REGION Network 5: Call production data cycle timer
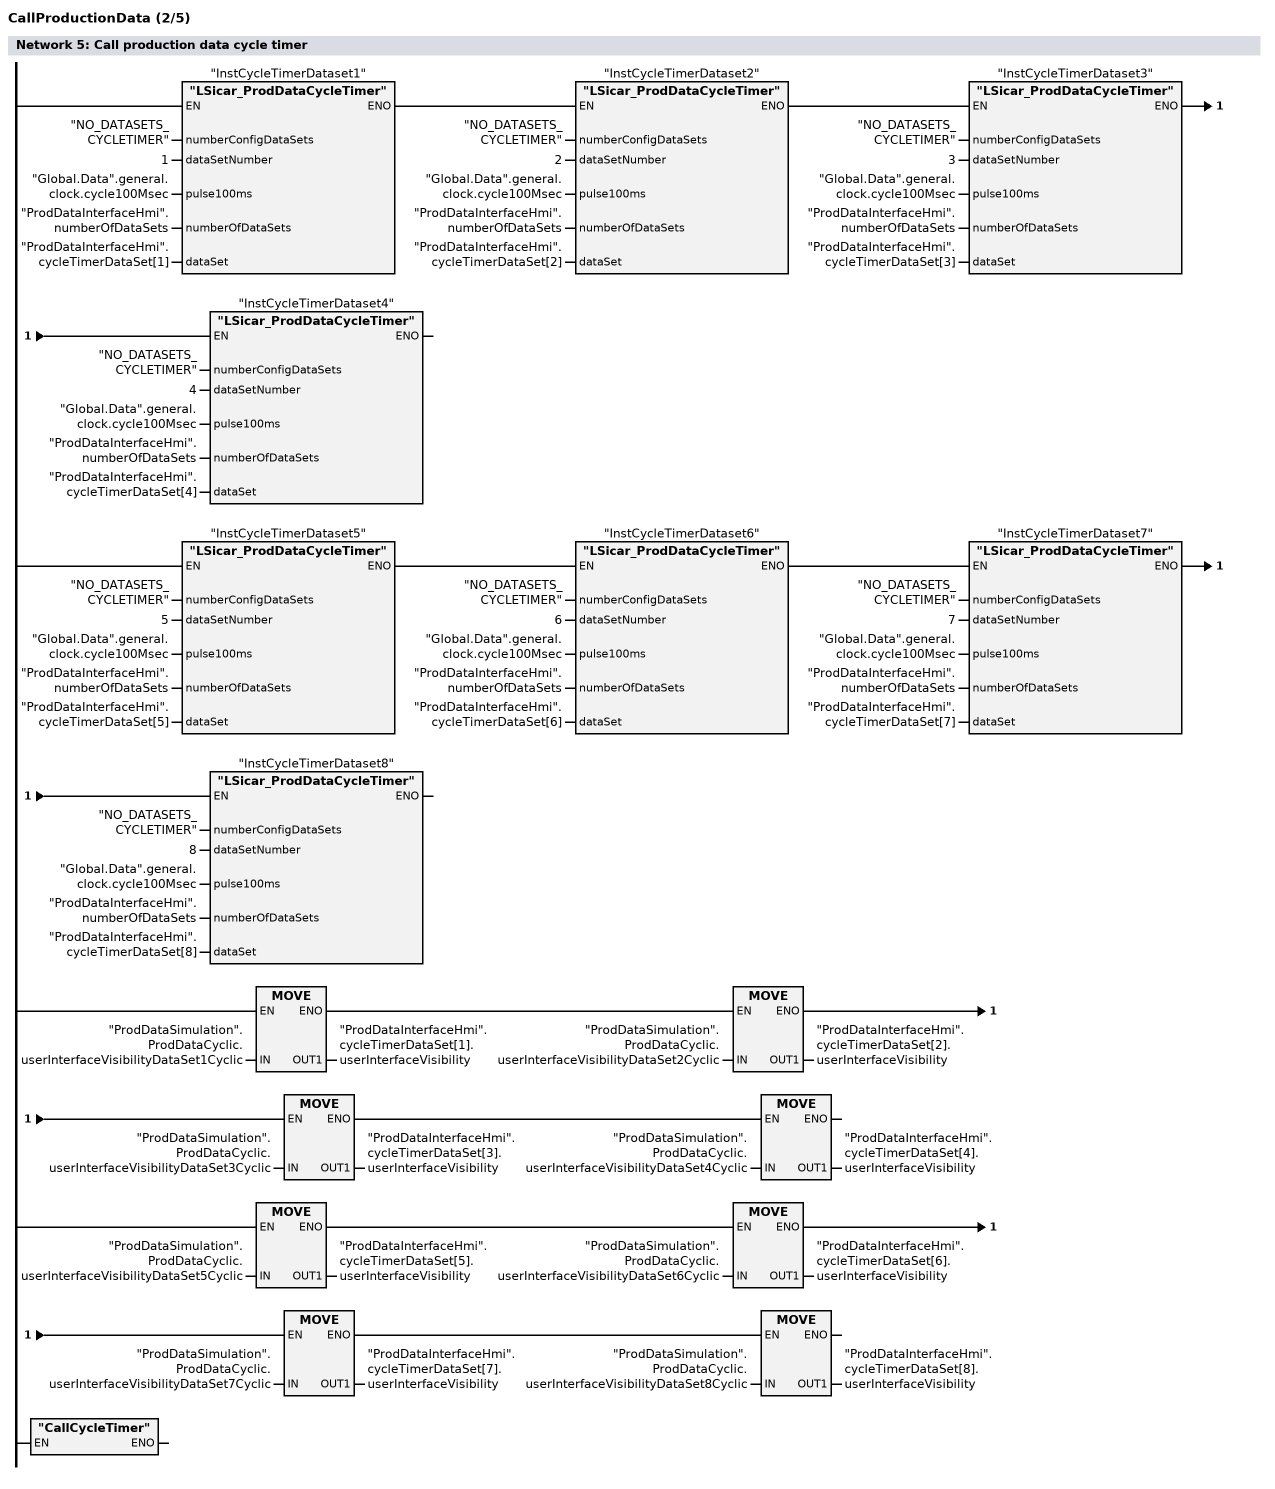
   RUNG wire#powerrail
      "InstCycleTimerDataset1"(numberConfigDataSets := "NO_DATASETS_CYCLETIMER", dataSetNumber := 1, pulse100ms := "Global.Data".general.clock.cycle100Msec, numberOfDataSets := "ProdDataInterfaceHmi".numberOfDataSets, dataSet := "ProdDataInterfaceHmi".cycleTimerDataSet[1])
      "InstCycleTimerDataset2"(numberConfigDataSets := "NO_DATASETS_CYCLETIMER", dataSetNumber := 2, pulse100ms := "Global.Data".general.clock.cycle100Msec, numberOfDataSets := "ProdDataInterfaceHmi".numberOfDataSets, dataSet := "ProdDataInterfaceHmi".cycleTimerDataSet[2])
      "InstCycleTimerDataset3"(numberConfigDataSets := "NO_DATASETS_CYCLETIMER", dataSetNumber := 3, pulse100ms := "Global.Data".general.clock.cycle100Msec, numberOfDataSets := "ProdDataInterfaceHmi".numberOfDataSets, dataSet := "ProdDataInterfaceHmi".cycleTimerDataSet[3])
      "InstCycleTimerDataset4"(numberConfigDataSets := "NO_DATASETS_CYCLETIMER", dataSetNumber := 4, pulse100ms := "Global.Data".general.clock.cycle100Msec, numberOfDataSets := "ProdDataInterfaceHmi".numberOfDataSets, dataSet := "ProdDataInterfaceHmi".cycleTimerDataSet[4])
   END_RUNG
   RUNG wire#powerrail
      "InstCycleTimerDataset5"(numberConfigDataSets := "NO_DATASETS_CYCLETIMER", dataSetNumber := 5, pulse100ms := "Global.Data".general.clock.cycle100Msec, numberOfDataSets := "ProdDataInterfaceHmi".numberOfDataSets, dataSet := "ProdDataInterfaceHmi".cycleTimerDataSet[5])
      "InstCycleTimerDataset6"(numberConfigDataSets := "NO_DATASETS_CYCLETIMER", dataSetNumber := 6, pulse100ms := "Global.Data".general.clock.cycle100Msec, numberOfDataSets := "ProdDataInterfaceHmi".numberOfDataSets, dataSet := "ProdDataInterfaceHmi".cycleTimerDataSet[6])
      "InstCycleTimerDataset7"(numberConfigDataSets := "NO_DATASETS_CYCLETIMER", dataSetNumber := 7, pulse100ms := "Global.Data".general.clock.cycle100Msec, numberOfDataSets := "ProdDataInterfaceHmi".numberOfDataSets, dataSet := "ProdDataInterfaceHmi".cycleTimerDataSet[7])
      "InstCycleTimerDataset8"(numberConfigDataSets := "NO_DATASETS_CYCLETIMER", dataSetNumber := 8, pulse100ms := "Global.Data".general.clock.cycle100Msec, numberOfDataSets := "ProdDataInterfaceHmi".numberOfDataSets, dataSet := "ProdDataInterfaceHmi".cycleTimerDataSet[8])
   END_RUNG
   RUNG wire#powerrail
      Move(in := "ProdDataSimulation".ProdDataCyclic.userInterfaceVisibilityDataSet1Cyclic, out1 => "ProdDataInterfaceHmi".cycleTimerDataSet[1].userInterfaceVisibility)
      Move(in := "ProdDataSimulation".ProdDataCyclic.userInterfaceVisibilityDataSet2Cyclic, out1 => "ProdDataInterfaceHmi".cycleTimerDataSet[2].userInterfaceVisibility)
      Move(in := "ProdDataSimulation".ProdDataCyclic.userInterfaceVisibilityDataSet3Cyclic, out1 => "ProdDataInterfaceHmi".cycleTimerDataSet[3].userInterfaceVisibility)
      Move(in := "ProdDataSimulation".ProdDataCyclic.userInterfaceVisibilityDataSet4Cyclic, out1 => "ProdDataInterfaceHmi".cycleTimerDataSet[4].userInterfaceVisibility)
   END_RUNG
   RUNG wire#powerrail
      Move(in := "ProdDataSimulation".ProdDataCyclic.userInterfaceVisibilityDataSet5Cyclic, out1 => "ProdDataInterfaceHmi".cycleTimerDataSet[5].userInterfaceVisibility)
      Move(in := "ProdDataSimulation".ProdDataCyclic.userInterfaceVisibilityDataSet6Cyclic, out1 => "ProdDataInterfaceHmi".cycleTimerDataSet[6].userInterfaceVisibility)
      Move(in := "ProdDataSimulation".ProdDataCyclic.userInterfaceVisibilityDataSet7Cyclic, out1 => "ProdDataInterfaceHmi".cycleTimerDataSet[7].userInterfaceVisibility)
      Move(in := "ProdDataSimulation".ProdDataCyclic.userInterfaceVisibilityDataSet8Cyclic, out1 => "ProdDataInterfaceHmi".cycleTimerDataSet[8].userInterfaceVisibility)
   END_RUNG
   RUNG wire#powerrail
      "CallCycleTimer"()
   END_RUNG
   // the same network as SCL:
   "InstCycleTimerDataset1"(numberConfigDataSets := "NO_DATASETS_CYCLETIMER",   // "LSicar_ProdDataCycleTimer"
                           dataSetNumber := 1,
                           pulse100ms := "Global.Data".general.clock.cycle100Msec,
                           numberOfDataSets := "ProdDataInterfaceHmi".numberOfDataSets,
                           dataSet := "ProdDataInterfaceHmi".cycleTimerDataSet[1],
                           ENO => #_w1);
   "InstCycleTimerDataset2"(EN := #_w1,   // "LSicar_ProdDataCycleTimer"
                           numberConfigDataSets := "NO_DATASETS_CYCLETIMER",
                           dataSetNumber := 2,
                           pulse100ms := "Global.Data".general.clock.cycle100Msec,
                           numberOfDataSets := "ProdDataInterfaceHmi".numberOfDataSets,
                           dataSet := "ProdDataInterfaceHmi".cycleTimerDataSet[2],
                           ENO => #_w2);
   "InstCycleTimerDataset3"(EN := #_w2,   // "LSicar_ProdDataCycleTimer"
                           numberConfigDataSets := "NO_DATASETS_CYCLETIMER",
                           dataSetNumber := 3,
                           pulse100ms := "Global.Data".general.clock.cycle100Msec,
                           numberOfDataSets := "ProdDataInterfaceHmi".numberOfDataSets,
                           dataSet := "ProdDataInterfaceHmi".cycleTimerDataSet[3],
                           ENO => #_w3);
   IF #_w3 THEN
       "InstCycleTimerDataset4"(numberConfigDataSets := "NO_DATASETS_CYCLETIMER",   // "LSicar_ProdDataCycleTimer"
                               dataSetNumber := 4,
                               pulse100ms := "Global.Data".general.clock.cycle100Msec,
                               numberOfDataSets := "ProdDataInterfaceHmi".numberOfDataSets,
                               dataSet := "ProdDataInterfaceHmi".cycleTimerDataSet[4]);
   END_IF;
   "InstCycleTimerDataset5"(numberConfigDataSets := "NO_DATASETS_CYCLETIMER",   // "LSicar_ProdDataCycleTimer"
                           dataSetNumber := 5,
                           pulse100ms := "Global.Data".general.clock.cycle100Msec,
                           numberOfDataSets := "ProdDataInterfaceHmi".numberOfDataSets,
                           dataSet := "ProdDataInterfaceHmi".cycleTimerDataSet[5],
                           ENO => #_w4);
   "InstCycleTimerDataset6"(EN := #_w4,   // "LSicar_ProdDataCycleTimer"
                           numberConfigDataSets := "NO_DATASETS_CYCLETIMER",
                           dataSetNumber := 6,
                           pulse100ms := "Global.Data".general.clock.cycle100Msec,
                           numberOfDataSets := "ProdDataInterfaceHmi".numberOfDataSets,
                           dataSet := "ProdDataInterfaceHmi".cycleTimerDataSet[6],
                           ENO => #_w5);
   "InstCycleTimerDataset7"(EN := #_w5,   // "LSicar_ProdDataCycleTimer"
                           numberConfigDataSets := "NO_DATASETS_CYCLETIMER",
                           dataSetNumber := 7,
                           pulse100ms := "Global.Data".general.clock.cycle100Msec,
                           numberOfDataSets := "ProdDataInterfaceHmi".numberOfDataSets,
                           dataSet := "ProdDataInterfaceHmi".cycleTimerDataSet[7],
                           ENO => #_w6);
   IF #_w6 THEN
       "InstCycleTimerDataset8"(numberConfigDataSets := "NO_DATASETS_CYCLETIMER",   // "LSicar_ProdDataCycleTimer"
                               dataSetNumber := 8,
                               pulse100ms := "Global.Data".general.clock.cycle100Msec,
                               numberOfDataSets := "ProdDataInterfaceHmi".numberOfDataSets,
                               dataSet := "ProdDataInterfaceHmi".cycleTimerDataSet[8]);
   END_IF;
   "ProdDataInterfaceHmi".cycleTimerDataSet[1].userInterfaceVisibility := "ProdDataSimulation".ProdDataCyclic.userInterfaceVisibilityDataSet1Cyclic;
   "ProdDataInterfaceHmi".cycleTimerDataSet[2].userInterfaceVisibility := "ProdDataSimulation".ProdDataCyclic.userInterfaceVisibilityDataSet2Cyclic;
   "ProdDataInterfaceHmi".cycleTimerDataSet[3].userInterfaceVisibility := "ProdDataSimulation".ProdDataCyclic.userInterfaceVisibilityDataSet3Cyclic;
   "ProdDataInterfaceHmi".cycleTimerDataSet[4].userInterfaceVisibility := "ProdDataSimulation".ProdDataCyclic.userInterfaceVisibilityDataSet4Cyclic;
   "ProdDataInterfaceHmi".cycleTimerDataSet[5].userInterfaceVisibility := "ProdDataSimulation".ProdDataCyclic.userInterfaceVisibilityDataSet5Cyclic;
   "ProdDataInterfaceHmi".cycleTimerDataSet[6].userInterfaceVisibility := "ProdDataSimulation".ProdDataCyclic.userInterfaceVisibilityDataSet6Cyclic;
   "ProdDataInterfaceHmi".cycleTimerDataSet[7].userInterfaceVisibility := "ProdDataSimulation".ProdDataCyclic.userInterfaceVisibilityDataSet7Cyclic;
   "ProdDataInterfaceHmi".cycleTimerDataSet[8].userInterfaceVisibility := "ProdDataSimulation".ProdDataCyclic.userInterfaceVisibilityDataSet8Cyclic;
   "CallCycleTimer"();
END_REGION

REGION Network 6: Beispiel: Limit Value 1..2 / Call production data limit values
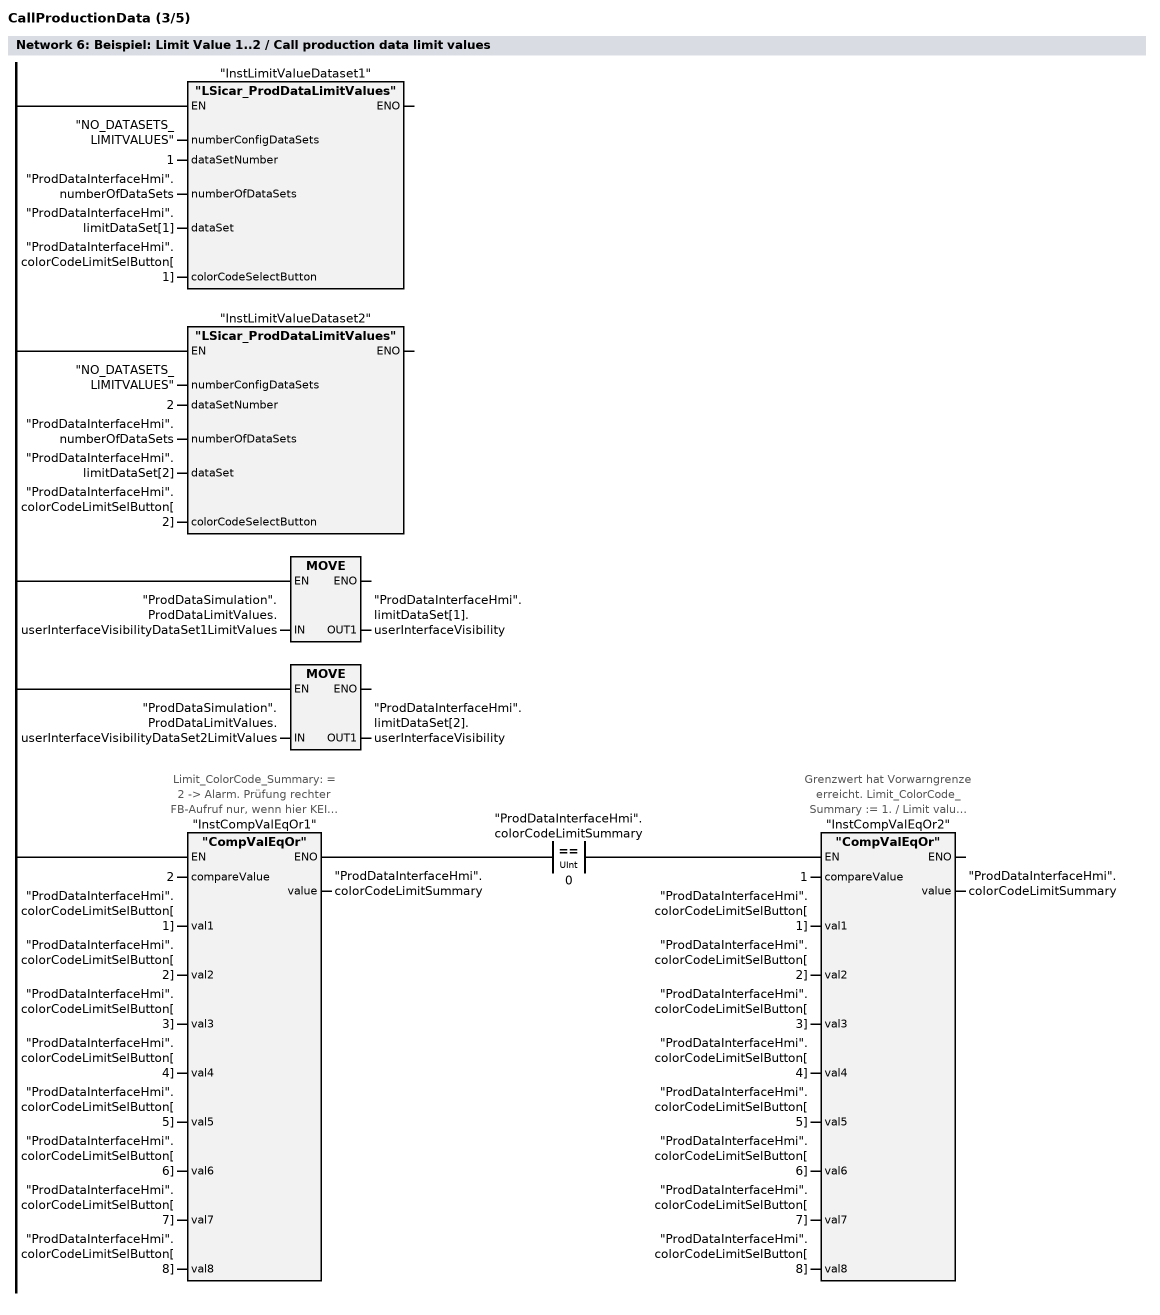
   RUNG wire#powerrail
      "InstLimitValueDataset1"(numberConfigDataSets := "NO_DATASETS_LIMITVALUES", dataSetNumber := 1, numberOfDataSets := "ProdDataInterfaceHmi".numberOfDataSets, dataSet := "ProdDataInterfaceHmi".limitDataSet[1], colorCodeSelectButton := "ProdDataInterfaceHmi".colorCodeLimitSelButton[1])
   END_RUNG
   RUNG wire#powerrail
      "InstLimitValueDataset2"(numberConfigDataSets := "NO_DATASETS_LIMITVALUES", dataSetNumber := 2, numberOfDataSets := "ProdDataInterfaceHmi".numberOfDataSets, dataSet := "ProdDataInterfaceHmi".limitDataSet[2], colorCodeSelectButton := "ProdDataInterfaceHmi".colorCodeLimitSelButton[2])
   END_RUNG
   RUNG wire#powerrail
      Move(in := "ProdDataSimulation".ProdDataLimitValues.userInterfaceVisibilityDataSet1LimitValues, out1 => "ProdDataInterfaceHmi".limitDataSet[1].userInterfaceVisibility)
   END_RUNG
   RUNG wire#powerrail
      Move(in := "ProdDataSimulation".ProdDataLimitValues.userInterfaceVisibilityDataSet2LimitValues, out1 => "ProdDataInterfaceHmi".limitDataSet[2].userInterfaceVisibility)
   END_RUNG
   RUNG wire#powerrail
      "InstCompValEqOr1"(compareValue := 2, val1 := "ProdDataInterfaceHmi".colorCodeLimitSelButton[1], val2 := "ProdDataInterfaceHmi".colorCodeLimitSelButton[2], val3 := "ProdDataInterfaceHmi".colorCodeLimitSelButton[3], val4 := "ProdDataInterfaceHmi".colorCodeLimitSelButton[4], val5 := "ProdDataInterfaceHmi".colorCodeLimitSelButton[5], val6 := "ProdDataInterfaceHmi".colorCodeLimitSelButton[6], val7 := "ProdDataInterfaceHmi".colorCodeLimitSelButton[7], val8 := "ProdDataInterfaceHmi".colorCodeLimitSelButton[8], value => "ProdDataInterfaceHmi".colorCodeLimitSummary)   // Limit_ColorCode_Summary: = 2 -> Alarm. Prüfung rechter FB-Aufruf nur, wenn hier KEIN Alarm (VALUE = 0) ansteht; Alarm ist höher prior. / Limit value = 2 -> Alarm. Limit_ColorCode_Summary := 2. Call right block only, if NO alarm (VALUE = 0) is pending here; alarm is higher prior.
      { S7_Templates := "SrcType := UInt" } EQ_Contact(in1 := "ProdDataInterfaceHmi".colorCodeLimitSummary, in2 := 0)
      "InstCompValEqOr2"(compareValue := 1, val1 := "ProdDataInterfaceHmi".colorCodeLimitSelButton[1], val2 := "ProdDataInterfaceHmi".colorCodeLimitSelButton[2], val3 := "ProdDataInterfaceHmi".colorCodeLimitSelButton[3], val4 := "ProdDataInterfaceHmi".colorCodeLimitSelButton[4], val5 := "ProdDataInterfaceHmi".colorCodeLimitSelButton[5], val6 := "ProdDataInterfaceHmi".colorCodeLimitSelButton[6], val7 := "ProdDataInterfaceHmi".colorCodeLimitSelButton[7], val8 := "ProdDataInterfaceHmi".colorCodeLimitSelButton[8], value => "ProdDataInterfaceHmi".colorCodeLimitSummary)   // Grenzwert hat Vorwarngrenze erreicht. Limit_ColorCode_Summary := 1. / Limit value <= Prewarn value. Limit_ColorCode_Summary := 1.
   END_RUNG
   // the same network as SCL:
   "InstLimitValueDataset1"(numberConfigDataSets := "NO_DATASETS_LIMITVALUES",   // "LSicar_ProdDataLimitValues"
                           dataSetNumber := 1,
                           numberOfDataSets := "ProdDataInterfaceHmi".numberOfDataSets,
                           dataSet := "ProdDataInterfaceHmi".limitDataSet[1],
                           colorCodeSelectButton := "ProdDataInterfaceHmi".colorCodeLimitSelButton[1]);
   "InstLimitValueDataset2"(numberConfigDataSets := "NO_DATASETS_LIMITVALUES",   // "LSicar_ProdDataLimitValues"
                           dataSetNumber := 2,
                           numberOfDataSets := "ProdDataInterfaceHmi".numberOfDataSets,
                           dataSet := "ProdDataInterfaceHmi".limitDataSet[2],
                           colorCodeSelectButton := "ProdDataInterfaceHmi".colorCodeLimitSelButton[2]);
   "ProdDataInterfaceHmi".limitDataSet[1].userInterfaceVisibility := "ProdDataSimulation".ProdDataLimitValues.userInterfaceVisibilityDataSet1LimitValues;
   "ProdDataInterfaceHmi".limitDataSet[2].userInterfaceVisibility := "ProdDataSimulation".ProdDataLimitValues.userInterfaceVisibilityDataSet2LimitValues;
   "InstCompValEqOr1"(compareValue := 2,   // "CompValEqOr": Limit_ColorCode_Summary: = 2 -> Alarm. Prüfung rechter FB-Aufruf nur, wenn hier KEIN Alarm (VALUE = 0) ansteht; Alarm ist höher prior. / Limit value = 2 -> Alarm. Limit_ColorCode_Summary := 2. Call right block only, if NO alarm (VALUE = 0) is pending here; alarm is higher prior.
                      val1 := "ProdDataInterfaceHmi".colorCodeLimitSelButton[1],
                      val2 := "ProdDataInterfaceHmi".colorCodeLimitSelButton[2],
                      val3 := "ProdDataInterfaceHmi".colorCodeLimitSelButton[3],
                      val4 := "ProdDataInterfaceHmi".colorCodeLimitSelButton[4],
                      val5 := "ProdDataInterfaceHmi".colorCodeLimitSelButton[5],
                      val6 := "ProdDataInterfaceHmi".colorCodeLimitSelButton[6],
                      val7 := "ProdDataInterfaceHmi".colorCodeLimitSelButton[7],
                      val8 := "ProdDataInterfaceHmi".colorCodeLimitSelButton[8],
                      value => "ProdDataInterfaceHmi".colorCodeLimitSummary,
                      ENO => #_w1);
   IF #_w1 AND ("ProdDataInterfaceHmi".colorCodeLimitSummary = 0) THEN
       "InstCompValEqOr2"(compareValue := 1,   // "CompValEqOr": Grenzwert hat Vorwarngrenze erreicht. Limit_ColorCode_Summary := 1. / Limit value <= Prewarn value. Limit_ColorCode_Summary := 1.
                          val1 := "ProdDataInterfaceHmi".colorCodeLimitSelButton[1],
                          val2 := "ProdDataInterfaceHmi".colorCodeLimitSelButton[2],
                          val3 := "ProdDataInterfaceHmi".colorCodeLimitSelButton[3],
                          val4 := "ProdDataInterfaceHmi".colorCodeLimitSelButton[4],
                          val5 := "ProdDataInterfaceHmi".colorCodeLimitSelButton[5],
                          val6 := "ProdDataInterfaceHmi".colorCodeLimitSelButton[6],
                          val7 := "ProdDataInterfaceHmi".colorCodeLimitSelButton[7],
                          val8 := "ProdDataInterfaceHmi".colorCodeLimitSelButton[8],
                          value => "ProdDataInterfaceHmi".colorCodeLimitSummary);
   END_IF;
END_REGION

REGION Network 7: Beispiel: Shift Counter 1..2 / Call production data shift counter
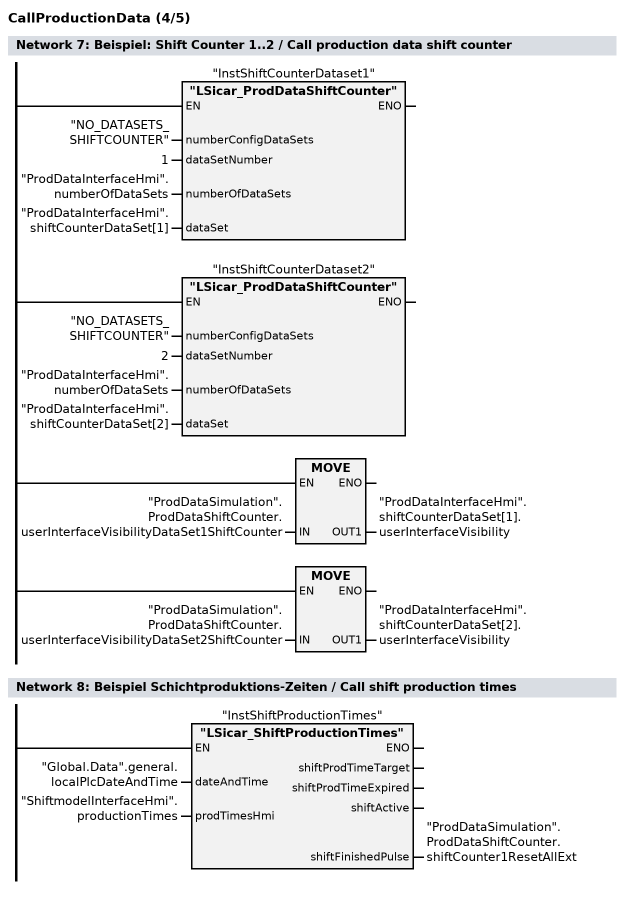
   RUNG wire#powerrail
      "InstShiftCounterDataset1"(numberConfigDataSets := "NO_DATASETS_SHIFTCOUNTER", dataSetNumber := 1, numberOfDataSets := "ProdDataInterfaceHmi".numberOfDataSets, dataSet := "ProdDataInterfaceHmi".shiftCounterDataSet[1])
   END_RUNG
   RUNG wire#powerrail
      "InstShiftCounterDataset2"(numberConfigDataSets := "NO_DATASETS_SHIFTCOUNTER", dataSetNumber := 2, numberOfDataSets := "ProdDataInterfaceHmi".numberOfDataSets, dataSet := "ProdDataInterfaceHmi".shiftCounterDataSet[2])
   END_RUNG
   RUNG wire#powerrail
      Move(in := "ProdDataSimulation".ProdDataShiftCounter.userInterfaceVisibilityDataSet1ShiftCounter, out1 => "ProdDataInterfaceHmi".shiftCounterDataSet[1].userInterfaceVisibility)
   END_RUNG
   RUNG wire#powerrail
      Move(in := "ProdDataSimulation".ProdDataShiftCounter.userInterfaceVisibilityDataSet2ShiftCounter, out1 => "ProdDataInterfaceHmi".shiftCounterDataSet[2].userInterfaceVisibility)
   END_RUNG
   // the same network as SCL:
   "InstShiftCounterDataset1"(numberConfigDataSets := "NO_DATASETS_SHIFTCOUNTER",   // "LSicar_ProdDataShiftCounter"
                           dataSetNumber := 1,
                           numberOfDataSets := "ProdDataInterfaceHmi".numberOfDataSets,
                           dataSet := "ProdDataInterfaceHmi".shiftCounterDataSet[1]);
   "InstShiftCounterDataset2"(numberConfigDataSets := "NO_DATASETS_SHIFTCOUNTER",   // "LSicar_ProdDataShiftCounter"
                           dataSetNumber := 2,
                           numberOfDataSets := "ProdDataInterfaceHmi".numberOfDataSets,
                           dataSet := "ProdDataInterfaceHmi".shiftCounterDataSet[2]);
   "ProdDataInterfaceHmi".shiftCounterDataSet[1].userInterfaceVisibility := "ProdDataSimulation".ProdDataShiftCounter.userInterfaceVisibilityDataSet1ShiftCounter;
   "ProdDataInterfaceHmi".shiftCounterDataSet[2].userInterfaceVisibility := "ProdDataSimulation".ProdDataShiftCounter.userInterfaceVisibilityDataSet2ShiftCounter;
END_REGION

REGION Network 8: Beispiel Schichtproduktions-Zeiten / Call shift production times
   RUNG wire#powerrail
      "InstShiftProductionTimes"(dateAndTime := "Global.Data".general.localPlcDateAndTime, prodTimesHmi := "ShiftmodelInterfaceHmi".productionTimes, shiftProdTimeTarget =>, shiftProdTimeExpired =>, shiftActive =>, shiftFinishedPulse => "ProdDataSimulation".ProdDataShiftCounter.shiftCounter1ResetAllExt)
   END_RUNG
   // the same network as SCL:
   "InstShiftProductionTimes"(dateAndTime := "Global.Data".general.localPlcDateAndTime,   // "LSicar_ShiftProductionTimes"
                           prodTimesHmi := "ShiftmodelInterfaceHmi".productionTimes,
                           shiftFinishedPulse => "ProdDataSimulation".ProdDataShiftCounter.shiftCounter1ResetAllExt);
END_REGION

REGION Network 9: Beispiel: Shift Counter 1..2 + OEE + Trend / Call production data shift counter OEE
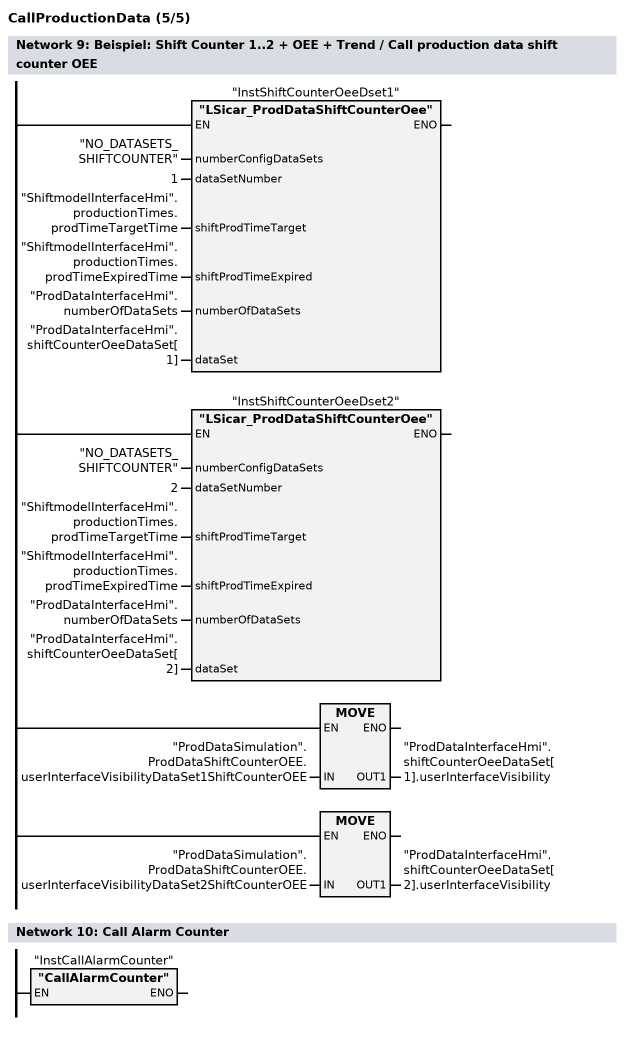
   RUNG wire#powerrail
      "InstShiftCounterOeeDset1"(numberConfigDataSets := "NO_DATASETS_SHIFTCOUNTER", dataSetNumber := 1, shiftProdTimeTarget := "ShiftmodelInterfaceHmi".productionTimes.prodTimeTargetTime, shiftProdTimeExpired := "ShiftmodelInterfaceHmi".productionTimes.prodTimeExpiredTime, numberOfDataSets := "ProdDataInterfaceHmi".numberOfDataSets, dataSet := "ProdDataInterfaceHmi".shiftCounterOeeDataSet[1])
   END_RUNG
   RUNG wire#powerrail
      "InstShiftCounterOeeDset2"(numberConfigDataSets := "NO_DATASETS_SHIFTCOUNTER", dataSetNumber := 2, shiftProdTimeTarget := "ShiftmodelInterfaceHmi".productionTimes.prodTimeTargetTime, shiftProdTimeExpired := "ShiftmodelInterfaceHmi".productionTimes.prodTimeExpiredTime, numberOfDataSets := "ProdDataInterfaceHmi".numberOfDataSets, dataSet := "ProdDataInterfaceHmi".shiftCounterOeeDataSet[2])
   END_RUNG
   RUNG wire#powerrail
      Move(in := "ProdDataSimulation".ProdDataShiftCounterOEE.userInterfaceVisibilityDataSet1ShiftCounterOEE, out1 => "ProdDataInterfaceHmi".shiftCounterOeeDataSet[1].userInterfaceVisibility)
   END_RUNG
   RUNG wire#powerrail
      Move(in := "ProdDataSimulation".ProdDataShiftCounterOEE.userInterfaceVisibilityDataSet2ShiftCounterOEE, out1 => "ProdDataInterfaceHmi".shiftCounterOeeDataSet[2].userInterfaceVisibility)
   END_RUNG
   // the same network as SCL:
   "InstShiftCounterOeeDset1"(numberConfigDataSets := "NO_DATASETS_SHIFTCOUNTER",   // "LSicar_ProdDataShiftCounterOee"
                           dataSetNumber := 1,
                           shiftProdTimeTarget := "ShiftmodelInterfaceHmi".productionTimes.prodTimeTargetTime,
                           shiftProdTimeExpired := "ShiftmodelInterfaceHmi".productionTimes.prodTimeExpiredTime,
                           numberOfDataSets := "ProdDataInterfaceHmi".numberOfDataSets,
                           dataSet := "ProdDataInterfaceHmi".shiftCounterOeeDataSet[1]);
   "InstShiftCounterOeeDset2"(numberConfigDataSets := "NO_DATASETS_SHIFTCOUNTER",   // "LSicar_ProdDataShiftCounterOee"
                           dataSetNumber := 2,
                           shiftProdTimeTarget := "ShiftmodelInterfaceHmi".productionTimes.prodTimeTargetTime,
                           shiftProdTimeExpired := "ShiftmodelInterfaceHmi".productionTimes.prodTimeExpiredTime,
                           numberOfDataSets := "ProdDataInterfaceHmi".numberOfDataSets,
                           dataSet := "ProdDataInterfaceHmi".shiftCounterOeeDataSet[2]);
   "ProdDataInterfaceHmi".shiftCounterOeeDataSet[1].userInterfaceVisibility := "ProdDataSimulation".ProdDataShiftCounterOEE.userInterfaceVisibilityDataSet1ShiftCounterOEE;
   "ProdDataInterfaceHmi".shiftCounterOeeDataSet[2].userInterfaceVisibility := "ProdDataSimulation".ProdDataShiftCounterOEE.userInterfaceVisibilityDataSet2ShiftCounterOEE;
END_REGION

REGION Network 10: Call Alarm Counter
   RUNG wire#powerrail
      "InstCallAlarmCounter"()
   END_RUNG
   // the same network as SCL:
   "InstCallAlarmCounter"();   // "CallAlarmCounter"
END_REGION
END_FUNCTION

FUNCTION "CallEnergy" : Void   // FC5, LAD
TITLE = CallEnergy
// Call of Demo EnergyMeter and Energy Efficient M for EEMM demonstration
// stored: IsIECCheckEnabled true, SetENOAutomatically true
BEGIN

REGION Network 1: BLOCK INFO HEADER
   // SIEMENS AG / (c)Copyright 2023
   // ------------------------------------------------------------------------------
   // Title:            CallEnergy (FC5)
   // Comment/Function: Call of Demo EnergyMeter and Energy Efficient M for EEMM demonstration
   // Library/Family:   Energy
   // Author:           SICAR
   // Tested with:      ---
   // Engineering:      TIA Portal V19
   // Restrictions:     -
   // Requirements:     ---
   // ------------------------------------------------------------------------------
   // Change log table:
   // Version  | Date       | Expert in charge       | Changes applied
   // ---------|------------|------------------------|------------------------------
   // 01.00.00 | 11.12.2023 | SICAR
   //                         First released version
END_REGION

REGION Network 2: Call: Demo EnergyMeter, Energy Efficient M
   // Call for EEM demonstration
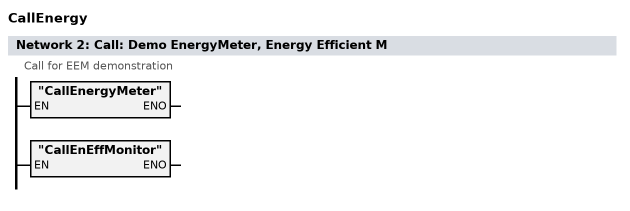
   RUNG wire#powerrail
      "CallEnergyMeter"()
   END_RUNG
   RUNG wire#powerrail
      "CallEnEffMonitor"()
   END_RUNG
   // the same network as SCL:
   "CallEnergyMeter"();
   "CallEnEffMonitor"();
END_REGION

REGION Network 3: Empty
END_REGION
END_FUNCTION

FUNCTION "SafetyState" : Void   // FC97, LAD
// stored: SetENOAutomatically true
   VAR CONSTANT
      TRUE : Bool := TRUE;
      FALSE : Bool;
   END_VAR
   VAR_TEMP   // added for the SCL form of the ladder/FBD networks
      _w1 : Bool;
   END_VAR
BEGIN

REGION Network 1: Stack Door Common Command#1
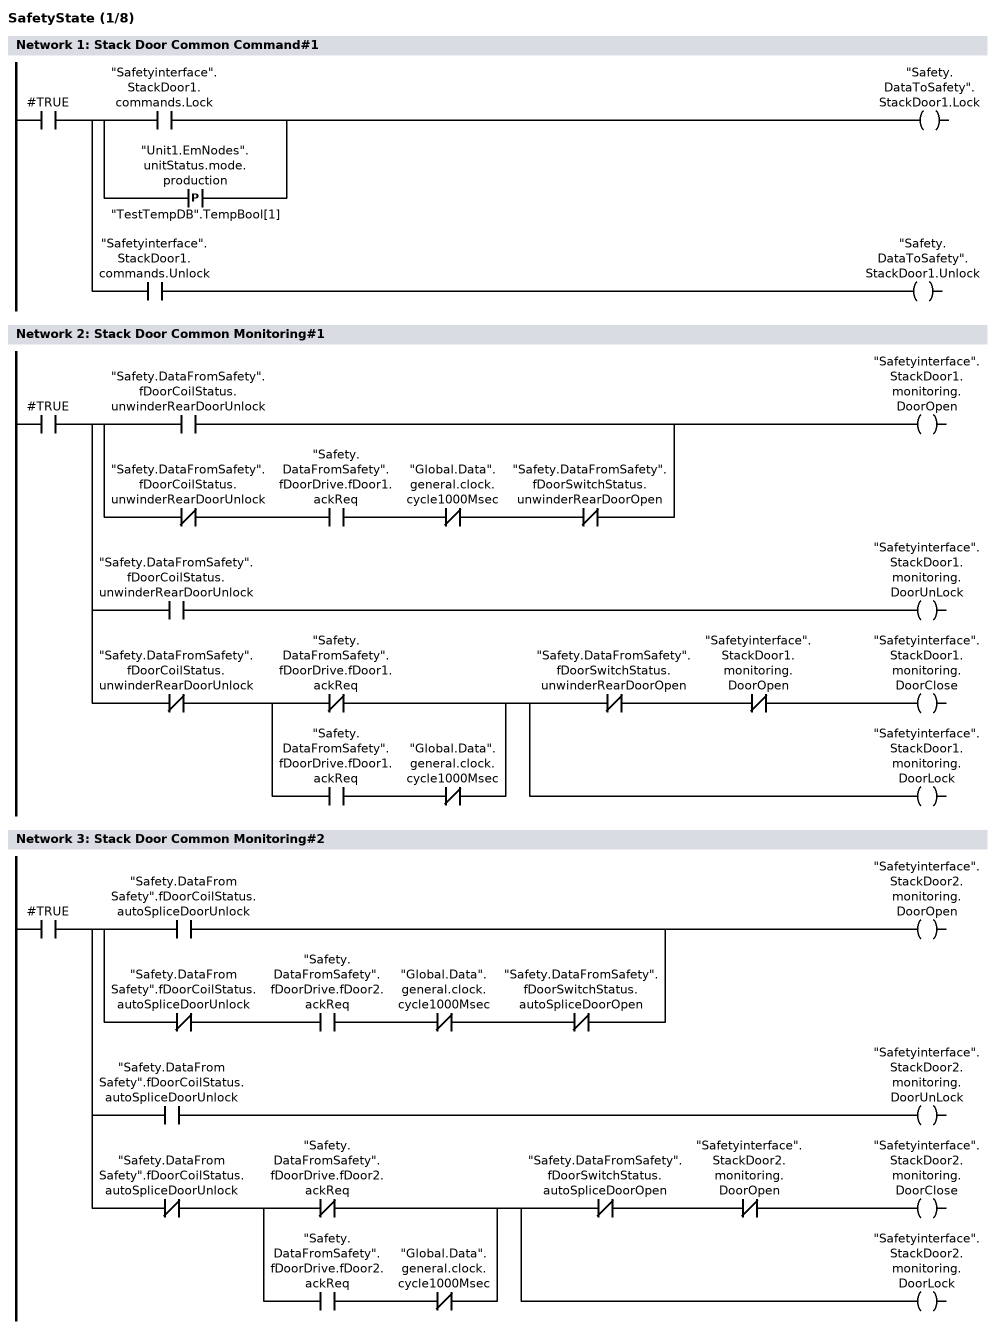
   RUNG wire#powerrail
      Contact( #TRUE )
      wire#w1
      Contact( "Safetyinterface".StackDoor1.commands.Lock )
      wire#w2
      Coil( "Safety.DataToSafety".StackDoor1.Lock )
   END_RUNG
   RUNG wire#w1
      P_Contact(operand := "Unit1.EmNodes".unitStatus.mode.production, bit := "TestTempDB".TempBool[1])
   END_RUNG wire#w2
   RUNG wire#w1
      Contact( "Safetyinterface".StackDoor1.commands.Unlock )
      Coil( "Safety.DataToSafety".StackDoor1.Unlock )
   END_RUNG
   // the same network as SCL:
   #_w1 := #TRUE AND "Unit1.EmNodes".unitStatus.mode.production AND NOT "TestTempDB".TempBool[1];   // rising edge of "Unit1.EmNodes".unitStatus.mode.production
   "TestTempDB".TempBool[1] := "Unit1.EmNodes".unitStatus.mode.production;
   "Safety.DataToSafety".StackDoor1.Lock := (#TRUE AND "Safetyinterface".StackDoor1.commands.Lock) OR #_w1;
   "Safety.DataToSafety".StackDoor1.Unlock := #TRUE AND "Safetyinterface".StackDoor1.commands.Unlock;
END_REGION

REGION Network 2: Stack Door Common Monitoring#1
   RUNG wire#powerrail
      Contact( #TRUE )
      wire#w1
      Contact( "Safety.DataFromSafety".fDoorCoilStatus.unwinderRearDoorUnlock )
      wire#w2
      Coil( "Safetyinterface".StackDoor1.monitoring.DoorOpen )
   END_RUNG
   RUNG wire#w1
      I_Contact( "Safety.DataFromSafety".fDoorCoilStatus.unwinderRearDoorUnlock )
      Contact( "Safety.DataFromSafety".fDoorDrive.fDoor1.ackReq )
      I_Contact( "Global.Data".general.clock.cycle1000Msec )
      I_Contact( "Safety.DataFromSafety".fDoorSwitchStatus.unwinderRearDoorOpen )
   END_RUNG wire#w2
   RUNG wire#w1
      Contact( "Safety.DataFromSafety".fDoorCoilStatus.unwinderRearDoorUnlock )
      Coil( "Safetyinterface".StackDoor1.monitoring.DoorUnLock )
   END_RUNG
   RUNG wire#w1
      I_Contact( "Safety.DataFromSafety".fDoorCoilStatus.unwinderRearDoorUnlock )
      wire#w3
      I_Contact( "Safety.DataFromSafety".fDoorDrive.fDoor1.ackReq )
      wire#w4
      I_Contact( "Safety.DataFromSafety".fDoorSwitchStatus.unwinderRearDoorOpen )
      I_Contact( "Safetyinterface".StackDoor1.monitoring.DoorOpen )
      Coil( "Safetyinterface".StackDoor1.monitoring.DoorClose )
   END_RUNG
   RUNG wire#w3
      Contact( "Safety.DataFromSafety".fDoorDrive.fDoor1.ackReq )
      I_Contact( "Global.Data".general.clock.cycle1000Msec )
   END_RUNG wire#w4
   RUNG wire#w4
      Coil( "Safetyinterface".StackDoor1.monitoring.DoorLock )
   END_RUNG
   // the same network as SCL:
   "Safetyinterface".StackDoor1.monitoring.DoorOpen := #TRUE AND ("Safety.DataFromSafety".fDoorCoilStatus.unwinderRearDoorUnlock OR (NOT "Safety.DataFromSafety".fDoorCoilStatus.unwinderRearDoorUnlock AND "Safety.DataFromSafety".fDoorDrive.fDoor1.ackReq AND NOT "Global.Data".general.clock.cycle1000Msec AND NOT "Safety.DataFromSafety".fDoorSwitchStatus.unwinderRearDoorOpen));
   "Safetyinterface".StackDoor1.monitoring.DoorUnLock := #TRUE AND "Safety.DataFromSafety".fDoorCoilStatus.unwinderRearDoorUnlock;
   #_w1 := #TRUE AND NOT "Safety.DataFromSafety".fDoorCoilStatus.unwinderRearDoorUnlock AND (NOT "Safety.DataFromSafety".fDoorDrive.fDoor1.ackReq OR ("Safety.DataFromSafety".fDoorDrive.fDoor1.ackReq AND NOT "Global.Data".general.clock.cycle1000Msec));
   "Safetyinterface".StackDoor1.monitoring.DoorClose := #_w1 AND NOT "Safety.DataFromSafety".fDoorSwitchStatus.unwinderRearDoorOpen AND NOT "Safetyinterface".StackDoor1.monitoring.DoorOpen;
   "Safetyinterface".StackDoor1.monitoring.DoorLock := #_w1;
END_REGION

REGION Network 3: Stack Door Common Monitoring#2
   RUNG wire#powerrail
      Contact( #TRUE )
      wire#w1
      Contact( "Safety.DataFromSafety".fDoorCoilStatus.autoSpliceDoorUnlock )
      wire#w2
      Coil( "Safetyinterface".StackDoor2.monitoring.DoorOpen )
   END_RUNG
   RUNG wire#w1
      I_Contact( "Safety.DataFromSafety".fDoorCoilStatus.autoSpliceDoorUnlock )
      Contact( "Safety.DataFromSafety".fDoorDrive.fDoor2.ackReq )
      I_Contact( "Global.Data".general.clock.cycle1000Msec )
      I_Contact( "Safety.DataFromSafety".fDoorSwitchStatus.autoSpliceDoorOpen )
   END_RUNG wire#w2
   RUNG wire#w1
      Contact( "Safety.DataFromSafety".fDoorCoilStatus.autoSpliceDoorUnlock )
      Coil( "Safetyinterface".StackDoor2.monitoring.DoorUnLock )
   END_RUNG
   RUNG wire#w1
      I_Contact( "Safety.DataFromSafety".fDoorCoilStatus.autoSpliceDoorUnlock )
      wire#w3
      I_Contact( "Safety.DataFromSafety".fDoorDrive.fDoor2.ackReq )
      wire#w4
      I_Contact( "Safety.DataFromSafety".fDoorSwitchStatus.autoSpliceDoorOpen )
      I_Contact( "Safetyinterface".StackDoor2.monitoring.DoorOpen )
      Coil( "Safetyinterface".StackDoor2.monitoring.DoorClose )
   END_RUNG
   RUNG wire#w3
      Contact( "Safety.DataFromSafety".fDoorDrive.fDoor2.ackReq )
      I_Contact( "Global.Data".general.clock.cycle1000Msec )
   END_RUNG wire#w4
   RUNG wire#w4
      Coil( "Safetyinterface".StackDoor2.monitoring.DoorLock )
   END_RUNG
   // the same network as SCL:
   "Safetyinterface".StackDoor2.monitoring.DoorOpen := #TRUE AND ("Safety.DataFromSafety".fDoorCoilStatus.autoSpliceDoorUnlock OR (NOT "Safety.DataFromSafety".fDoorCoilStatus.autoSpliceDoorUnlock AND "Safety.DataFromSafety".fDoorDrive.fDoor2.ackReq AND NOT "Global.Data".general.clock.cycle1000Msec AND NOT "Safety.DataFromSafety".fDoorSwitchStatus.autoSpliceDoorOpen));
   "Safetyinterface".StackDoor2.monitoring.DoorUnLock := #TRUE AND "Safety.DataFromSafety".fDoorCoilStatus.autoSpliceDoorUnlock;
   #_w1 := #TRUE AND NOT "Safety.DataFromSafety".fDoorCoilStatus.autoSpliceDoorUnlock AND (NOT "Safety.DataFromSafety".fDoorDrive.fDoor2.ackReq OR ("Safety.DataFromSafety".fDoorDrive.fDoor2.ackReq AND NOT "Global.Data".general.clock.cycle1000Msec));
   "Safetyinterface".StackDoor2.monitoring.DoorClose := #_w1 AND NOT "Safety.DataFromSafety".fDoorSwitchStatus.autoSpliceDoorOpen AND NOT "Safetyinterface".StackDoor2.monitoring.DoorOpen;
   "Safetyinterface".StackDoor2.monitoring.DoorLock := #_w1;
END_REGION

REGION Network 4: Stack Door Common Monitoring#3
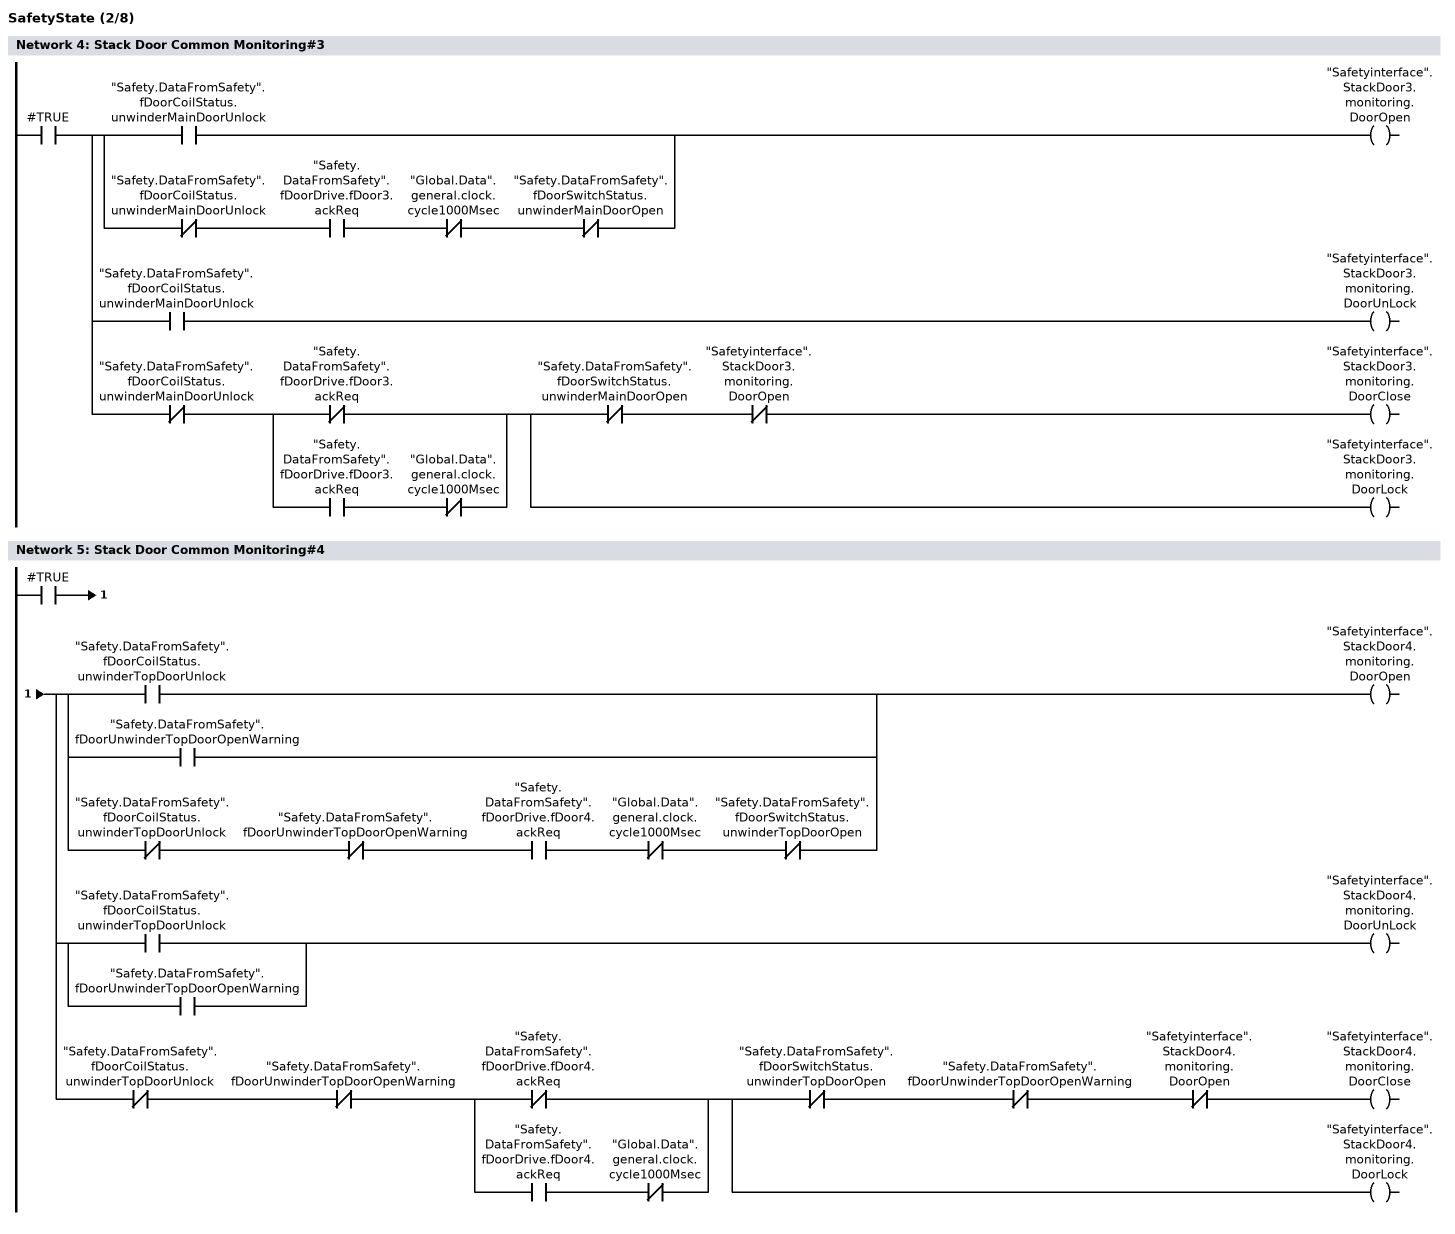
   RUNG wire#powerrail
      Contact( #TRUE )
      wire#w1
      Contact( "Safety.DataFromSafety".fDoorCoilStatus.unwinderMainDoorUnlock )
      wire#w2
      Coil( "Safetyinterface".StackDoor3.monitoring.DoorOpen )
   END_RUNG
   RUNG wire#w1
      I_Contact( "Safety.DataFromSafety".fDoorCoilStatus.unwinderMainDoorUnlock )
      Contact( "Safety.DataFromSafety".fDoorDrive.fDoor3.ackReq )
      I_Contact( "Global.Data".general.clock.cycle1000Msec )
      I_Contact( "Safety.DataFromSafety".fDoorSwitchStatus.unwinderMainDoorOpen )
   END_RUNG wire#w2
   RUNG wire#w1
      Contact( "Safety.DataFromSafety".fDoorCoilStatus.unwinderMainDoorUnlock )
      Coil( "Safetyinterface".StackDoor3.monitoring.DoorUnLock )
   END_RUNG
   RUNG wire#w1
      I_Contact( "Safety.DataFromSafety".fDoorCoilStatus.unwinderMainDoorUnlock )
      wire#w3
      I_Contact( "Safety.DataFromSafety".fDoorDrive.fDoor3.ackReq )
      wire#w4
      I_Contact( "Safety.DataFromSafety".fDoorSwitchStatus.unwinderMainDoorOpen )
      I_Contact( "Safetyinterface".StackDoor3.monitoring.DoorOpen )
      Coil( "Safetyinterface".StackDoor3.monitoring.DoorClose )
   END_RUNG
   RUNG wire#w3
      Contact( "Safety.DataFromSafety".fDoorDrive.fDoor3.ackReq )
      I_Contact( "Global.Data".general.clock.cycle1000Msec )
   END_RUNG wire#w4
   RUNG wire#w4
      Coil( "Safetyinterface".StackDoor3.monitoring.DoorLock )
   END_RUNG
   // the same network as SCL:
   "Safetyinterface".StackDoor3.monitoring.DoorOpen := #TRUE AND ("Safety.DataFromSafety".fDoorCoilStatus.unwinderMainDoorUnlock OR (NOT "Safety.DataFromSafety".fDoorCoilStatus.unwinderMainDoorUnlock AND "Safety.DataFromSafety".fDoorDrive.fDoor3.ackReq AND NOT "Global.Data".general.clock.cycle1000Msec AND NOT "Safety.DataFromSafety".fDoorSwitchStatus.unwinderMainDoorOpen));
   "Safetyinterface".StackDoor3.monitoring.DoorUnLock := #TRUE AND "Safety.DataFromSafety".fDoorCoilStatus.unwinderMainDoorUnlock;
   #_w1 := #TRUE AND NOT "Safety.DataFromSafety".fDoorCoilStatus.unwinderMainDoorUnlock AND (NOT "Safety.DataFromSafety".fDoorDrive.fDoor3.ackReq OR ("Safety.DataFromSafety".fDoorDrive.fDoor3.ackReq AND NOT "Global.Data".general.clock.cycle1000Msec));
   "Safetyinterface".StackDoor3.monitoring.DoorClose := #_w1 AND NOT "Safety.DataFromSafety".fDoorSwitchStatus.unwinderMainDoorOpen AND NOT "Safetyinterface".StackDoor3.monitoring.DoorOpen;
   "Safetyinterface".StackDoor3.monitoring.DoorLock := #_w1;
END_REGION

REGION Network 5: Stack Door Common Monitoring#4
   RUNG wire#powerrail
      Contact( #TRUE )
      wire#w1
      Contact( "Safety.DataFromSafety".fDoorCoilStatus.unwinderTopDoorUnlock )
      wire#w2
      Coil( "Safetyinterface".StackDoor4.monitoring.DoorOpen )
   END_RUNG
   RUNG wire#w1
      Contact( "Safety.DataFromSafety".fDoorUnwinderTopDoorOpenWarning )
   END_RUNG wire#w2
   RUNG wire#w1
      I_Contact( "Safety.DataFromSafety".fDoorCoilStatus.unwinderTopDoorUnlock )
      I_Contact( "Safety.DataFromSafety".fDoorUnwinderTopDoorOpenWarning )
      Contact( "Safety.DataFromSafety".fDoorDrive.fDoor4.ackReq )
      I_Contact( "Global.Data".general.clock.cycle1000Msec )
      I_Contact( "Safety.DataFromSafety".fDoorSwitchStatus.unwinderTopDoorOpen )
   END_RUNG wire#w2
   RUNG wire#w1
      Contact( "Safety.DataFromSafety".fDoorCoilStatus.unwinderTopDoorUnlock )
      wire#w3
      Coil( "Safetyinterface".StackDoor4.monitoring.DoorUnLock )
   END_RUNG
   RUNG wire#w1
      Contact( "Safety.DataFromSafety".fDoorUnwinderTopDoorOpenWarning )
   END_RUNG wire#w3
   RUNG wire#w1
      I_Contact( "Safety.DataFromSafety".fDoorCoilStatus.unwinderTopDoorUnlock )
      I_Contact( "Safety.DataFromSafety".fDoorUnwinderTopDoorOpenWarning )
      wire#w4
      I_Contact( "Safety.DataFromSafety".fDoorDrive.fDoor4.ackReq )
      wire#w5
      I_Contact( "Safety.DataFromSafety".fDoorSwitchStatus.unwinderTopDoorOpen )
      I_Contact( "Safety.DataFromSafety".fDoorUnwinderTopDoorOpenWarning )
      I_Contact( "Safetyinterface".StackDoor4.monitoring.DoorOpen )
      Coil( "Safetyinterface".StackDoor4.monitoring.DoorClose )
   END_RUNG
   RUNG wire#w4
      Contact( "Safety.DataFromSafety".fDoorDrive.fDoor4.ackReq )
      I_Contact( "Global.Data".general.clock.cycle1000Msec )
   END_RUNG wire#w5
   RUNG wire#w5
      Coil( "Safetyinterface".StackDoor4.monitoring.DoorLock )
   END_RUNG
   // the same network as SCL:
   "Safetyinterface".StackDoor4.monitoring.DoorOpen := #TRUE AND ("Safety.DataFromSafety".fDoorCoilStatus.unwinderTopDoorUnlock OR "Safety.DataFromSafety".fDoorUnwinderTopDoorOpenWarning OR (NOT "Safety.DataFromSafety".fDoorCoilStatus.unwinderTopDoorUnlock AND NOT "Safety.DataFromSafety".fDoorUnwinderTopDoorOpenWarning AND "Safety.DataFromSafety".fDoorDrive.fDoor4.ackReq AND NOT "Global.Data".general.clock.cycle1000Msec AND NOT "Safety.DataFromSafety".fDoorSwitchStatus.unwinderTopDoorOpen));
   "Safetyinterface".StackDoor4.monitoring.DoorUnLock := #TRUE AND ("Safety.DataFromSafety".fDoorCoilStatus.unwinderTopDoorUnlock OR "Safety.DataFromSafety".fDoorUnwinderTopDoorOpenWarning);
   #_w1 := #TRUE AND NOT "Safety.DataFromSafety".fDoorCoilStatus.unwinderTopDoorUnlock AND NOT "Safety.DataFromSafety".fDoorUnwinderTopDoorOpenWarning AND (NOT "Safety.DataFromSafety".fDoorDrive.fDoor4.ackReq OR ("Safety.DataFromSafety".fDoorDrive.fDoor4.ackReq AND NOT "Global.Data".general.clock.cycle1000Msec));
   "Safetyinterface".StackDoor4.monitoring.DoorClose := #_w1 AND NOT "Safety.DataFromSafety".fDoorSwitchStatus.unwinderTopDoorOpen AND NOT "Safety.DataFromSafety".fDoorUnwinderTopDoorOpenWarning AND NOT "Safetyinterface".StackDoor4.monitoring.DoorOpen;
   "Safetyinterface".StackDoor4.monitoring.DoorLock := #_w1;
END_REGION

REGION Network 6: Stack Door Common Monitoring#5
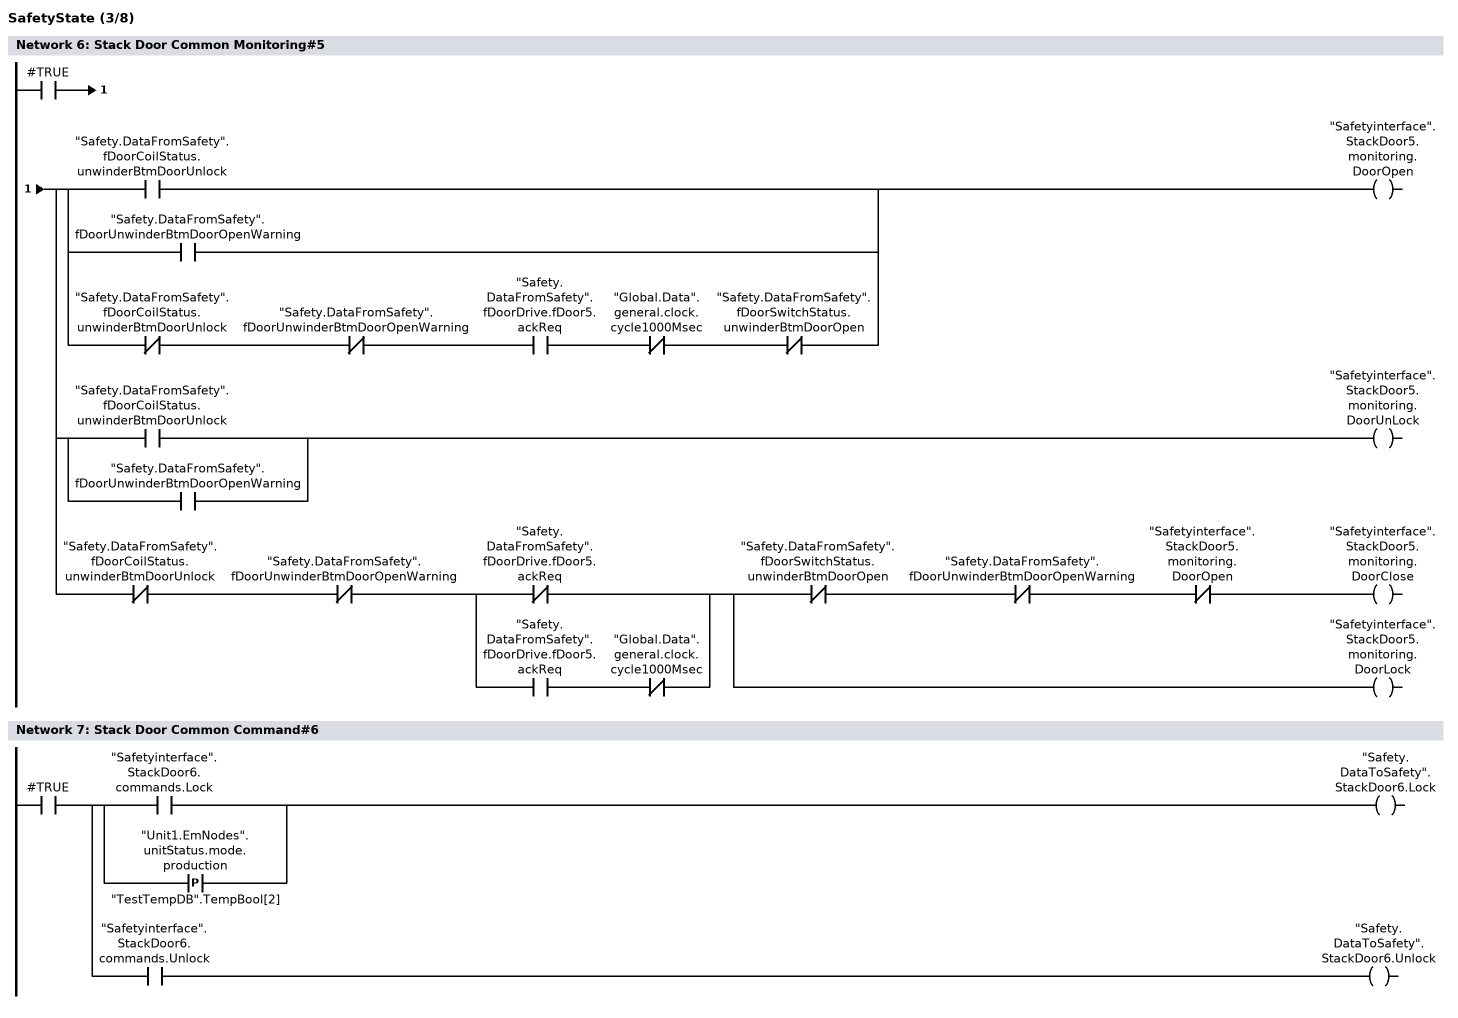
   RUNG wire#powerrail
      Contact( #TRUE )
      wire#w1
      Contact( "Safety.DataFromSafety".fDoorCoilStatus.unwinderBtmDoorUnlock )
      wire#w2
      Coil( "Safetyinterface".StackDoor5.monitoring.DoorOpen )
   END_RUNG
   RUNG wire#w1
      Contact( "Safety.DataFromSafety".fDoorUnwinderBtmDoorOpenWarning )
   END_RUNG wire#w2
   RUNG wire#w1
      I_Contact( "Safety.DataFromSafety".fDoorCoilStatus.unwinderBtmDoorUnlock )
      I_Contact( "Safety.DataFromSafety".fDoorUnwinderBtmDoorOpenWarning )
      Contact( "Safety.DataFromSafety".fDoorDrive.fDoor5.ackReq )
      I_Contact( "Global.Data".general.clock.cycle1000Msec )
      I_Contact( "Safety.DataFromSafety".fDoorSwitchStatus.unwinderBtmDoorOpen )
   END_RUNG wire#w2
   RUNG wire#w1
      Contact( "Safety.DataFromSafety".fDoorCoilStatus.unwinderBtmDoorUnlock )
      wire#w3
      Coil( "Safetyinterface".StackDoor5.monitoring.DoorUnLock )
   END_RUNG
   RUNG wire#w1
      Contact( "Safety.DataFromSafety".fDoorUnwinderBtmDoorOpenWarning )
   END_RUNG wire#w3
   RUNG wire#w1
      I_Contact( "Safety.DataFromSafety".fDoorCoilStatus.unwinderBtmDoorUnlock )
      I_Contact( "Safety.DataFromSafety".fDoorUnwinderBtmDoorOpenWarning )
      wire#w4
      I_Contact( "Safety.DataFromSafety".fDoorDrive.fDoor5.ackReq )
      wire#w5
      I_Contact( "Safety.DataFromSafety".fDoorSwitchStatus.unwinderBtmDoorOpen )
      I_Contact( "Safety.DataFromSafety".fDoorUnwinderBtmDoorOpenWarning )
      I_Contact( "Safetyinterface".StackDoor5.monitoring.DoorOpen )
      Coil( "Safetyinterface".StackDoor5.monitoring.DoorClose )
   END_RUNG
   RUNG wire#w4
      Contact( "Safety.DataFromSafety".fDoorDrive.fDoor5.ackReq )
      I_Contact( "Global.Data".general.clock.cycle1000Msec )
   END_RUNG wire#w5
   RUNG wire#w5
      Coil( "Safetyinterface".StackDoor5.monitoring.DoorLock )
   END_RUNG
   // the same network as SCL:
   "Safetyinterface".StackDoor5.monitoring.DoorOpen := #TRUE AND ("Safety.DataFromSafety".fDoorCoilStatus.unwinderBtmDoorUnlock OR "Safety.DataFromSafety".fDoorUnwinderBtmDoorOpenWarning OR (NOT "Safety.DataFromSafety".fDoorCoilStatus.unwinderBtmDoorUnlock AND NOT "Safety.DataFromSafety".fDoorUnwinderBtmDoorOpenWarning AND "Safety.DataFromSafety".fDoorDrive.fDoor5.ackReq AND NOT "Global.Data".general.clock.cycle1000Msec AND NOT "Safety.DataFromSafety".fDoorSwitchStatus.unwinderBtmDoorOpen));
   "Safetyinterface".StackDoor5.monitoring.DoorUnLock := #TRUE AND ("Safety.DataFromSafety".fDoorCoilStatus.unwinderBtmDoorUnlock OR "Safety.DataFromSafety".fDoorUnwinderBtmDoorOpenWarning);
   #_w1 := #TRUE AND NOT "Safety.DataFromSafety".fDoorCoilStatus.unwinderBtmDoorUnlock AND NOT "Safety.DataFromSafety".fDoorUnwinderBtmDoorOpenWarning AND (NOT "Safety.DataFromSafety".fDoorDrive.fDoor5.ackReq OR ("Safety.DataFromSafety".fDoorDrive.fDoor5.ackReq AND NOT "Global.Data".general.clock.cycle1000Msec));
   "Safetyinterface".StackDoor5.monitoring.DoorClose := #_w1 AND NOT "Safety.DataFromSafety".fDoorSwitchStatus.unwinderBtmDoorOpen AND NOT "Safety.DataFromSafety".fDoorUnwinderBtmDoorOpenWarning AND NOT "Safetyinterface".StackDoor5.monitoring.DoorOpen;
   "Safetyinterface".StackDoor5.monitoring.DoorLock := #_w1;
END_REGION

REGION Network 7: Stack Door Common Command#6
   RUNG wire#powerrail
      Contact( #TRUE )
      wire#w1
      Contact( "Safetyinterface".StackDoor6.commands.Lock )
      wire#w2
      Coil( "Safety.DataToSafety".StackDoor6.Lock )
   END_RUNG
   RUNG wire#w1
      P_Contact(operand := "Unit1.EmNodes".unitStatus.mode.production, bit := "TestTempDB".TempBool[2])
   END_RUNG wire#w2
   RUNG wire#w1
      Contact( "Safetyinterface".StackDoor6.commands.Unlock )
      Coil( "Safety.DataToSafety".StackDoor6.Unlock )
   END_RUNG
   // the same network as SCL:
   #_w1 := #TRUE AND "Unit1.EmNodes".unitStatus.mode.production AND NOT "TestTempDB".TempBool[2];   // rising edge of "Unit1.EmNodes".unitStatus.mode.production
   "TestTempDB".TempBool[2] := "Unit1.EmNodes".unitStatus.mode.production;
   "Safety.DataToSafety".StackDoor6.Lock := (#TRUE AND "Safetyinterface".StackDoor6.commands.Lock) OR #_w1;
   "Safety.DataToSafety".StackDoor6.Unlock := #TRUE AND "Safetyinterface".StackDoor6.commands.Unlock;
END_REGION

REGION Network 8: Stack Door Common Monitoring#6
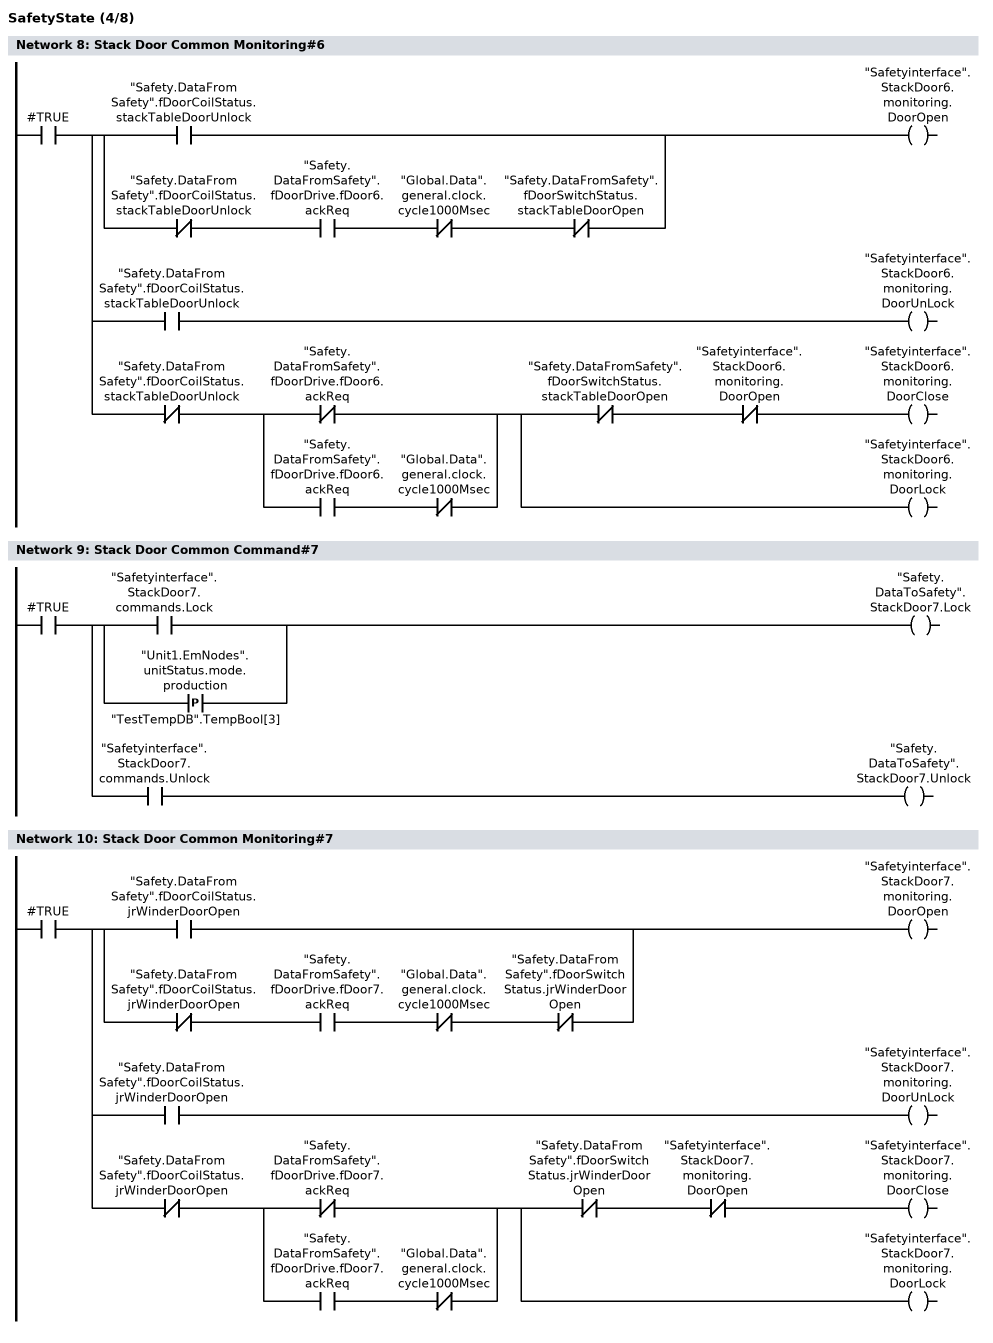
   RUNG wire#powerrail
      Contact( #TRUE )
      wire#w1
      Contact( "Safety.DataFromSafety".fDoorCoilStatus.stackTableDoorUnlock )
      wire#w2
      Coil( "Safetyinterface".StackDoor6.monitoring.DoorOpen )
   END_RUNG
   RUNG wire#w1
      I_Contact( "Safety.DataFromSafety".fDoorCoilStatus.stackTableDoorUnlock )
      Contact( "Safety.DataFromSafety".fDoorDrive.fDoor6.ackReq )
      I_Contact( "Global.Data".general.clock.cycle1000Msec )
      I_Contact( "Safety.DataFromSafety".fDoorSwitchStatus.stackTableDoorOpen )
   END_RUNG wire#w2
   RUNG wire#w1
      Contact( "Safety.DataFromSafety".fDoorCoilStatus.stackTableDoorUnlock )
      Coil( "Safetyinterface".StackDoor6.monitoring.DoorUnLock )
   END_RUNG
   RUNG wire#w1
      I_Contact( "Safety.DataFromSafety".fDoorCoilStatus.stackTableDoorUnlock )
      wire#w3
      I_Contact( "Safety.DataFromSafety".fDoorDrive.fDoor6.ackReq )
      wire#w4
      I_Contact( "Safety.DataFromSafety".fDoorSwitchStatus.stackTableDoorOpen )
      I_Contact( "Safetyinterface".StackDoor6.monitoring.DoorOpen )
      Coil( "Safetyinterface".StackDoor6.monitoring.DoorClose )
   END_RUNG
   RUNG wire#w3
      Contact( "Safety.DataFromSafety".fDoorDrive.fDoor6.ackReq )
      I_Contact( "Global.Data".general.clock.cycle1000Msec )
   END_RUNG wire#w4
   RUNG wire#w4
      Coil( "Safetyinterface".StackDoor6.monitoring.DoorLock )
   END_RUNG
   // the same network as SCL:
   "Safetyinterface".StackDoor6.monitoring.DoorOpen := #TRUE AND ("Safety.DataFromSafety".fDoorCoilStatus.stackTableDoorUnlock OR (NOT "Safety.DataFromSafety".fDoorCoilStatus.stackTableDoorUnlock AND "Safety.DataFromSafety".fDoorDrive.fDoor6.ackReq AND NOT "Global.Data".general.clock.cycle1000Msec AND NOT "Safety.DataFromSafety".fDoorSwitchStatus.stackTableDoorOpen));
   "Safetyinterface".StackDoor6.monitoring.DoorUnLock := #TRUE AND "Safety.DataFromSafety".fDoorCoilStatus.stackTableDoorUnlock;
   #_w1 := #TRUE AND NOT "Safety.DataFromSafety".fDoorCoilStatus.stackTableDoorUnlock AND (NOT "Safety.DataFromSafety".fDoorDrive.fDoor6.ackReq OR ("Safety.DataFromSafety".fDoorDrive.fDoor6.ackReq AND NOT "Global.Data".general.clock.cycle1000Msec));
   "Safetyinterface".StackDoor6.monitoring.DoorClose := #_w1 AND NOT "Safety.DataFromSafety".fDoorSwitchStatus.stackTableDoorOpen AND NOT "Safetyinterface".StackDoor6.monitoring.DoorOpen;
   "Safetyinterface".StackDoor6.monitoring.DoorLock := #_w1;
END_REGION

REGION Network 9: Stack Door Common Command#7
   RUNG wire#powerrail
      Contact( #TRUE )
      wire#w1
      Contact( "Safetyinterface".StackDoor7.commands.Lock )
      wire#w2
      Coil( "Safety.DataToSafety".StackDoor7.Lock )
   END_RUNG
   RUNG wire#w1
      P_Contact(operand := "Unit1.EmNodes".unitStatus.mode.production, bit := "TestTempDB".TempBool[3])
   END_RUNG wire#w2
   RUNG wire#w1
      Contact( "Safetyinterface".StackDoor7.commands.Unlock )
      Coil( "Safety.DataToSafety".StackDoor7.Unlock )
   END_RUNG
   // the same network as SCL:
   #_w1 := #TRUE AND "Unit1.EmNodes".unitStatus.mode.production AND NOT "TestTempDB".TempBool[3];   // rising edge of "Unit1.EmNodes".unitStatus.mode.production
   "TestTempDB".TempBool[3] := "Unit1.EmNodes".unitStatus.mode.production;
   "Safety.DataToSafety".StackDoor7.Lock := (#TRUE AND "Safetyinterface".StackDoor7.commands.Lock) OR #_w1;
   "Safety.DataToSafety".StackDoor7.Unlock := #TRUE AND "Safetyinterface".StackDoor7.commands.Unlock;
END_REGION

REGION Network 10: Stack Door Common Monitoring#7
   RUNG wire#powerrail
      Contact( #TRUE )
      wire#w1
      Contact( "Safety.DataFromSafety".fDoorCoilStatus.jrWinderDoorOpen )
      wire#w2
      Coil( "Safetyinterface".StackDoor7.monitoring.DoorOpen )
   END_RUNG
   RUNG wire#w1
      I_Contact( "Safety.DataFromSafety".fDoorCoilStatus.jrWinderDoorOpen )
      Contact( "Safety.DataFromSafety".fDoorDrive.fDoor7.ackReq )
      I_Contact( "Global.Data".general.clock.cycle1000Msec )
      I_Contact( "Safety.DataFromSafety".fDoorSwitchStatus.jrWinderDoorOpen )
   END_RUNG wire#w2
   RUNG wire#w1
      Contact( "Safety.DataFromSafety".fDoorCoilStatus.jrWinderDoorOpen )
      Coil( "Safetyinterface".StackDoor7.monitoring.DoorUnLock )
   END_RUNG
   RUNG wire#w1
      I_Contact( "Safety.DataFromSafety".fDoorCoilStatus.jrWinderDoorOpen )
      wire#w3
      I_Contact( "Safety.DataFromSafety".fDoorDrive.fDoor7.ackReq )
      wire#w4
      I_Contact( "Safety.DataFromSafety".fDoorSwitchStatus.jrWinderDoorOpen )
      I_Contact( "Safetyinterface".StackDoor7.monitoring.DoorOpen )
      Coil( "Safetyinterface".StackDoor7.monitoring.DoorClose )
   END_RUNG
   RUNG wire#w3
      Contact( "Safety.DataFromSafety".fDoorDrive.fDoor7.ackReq )
      I_Contact( "Global.Data".general.clock.cycle1000Msec )
   END_RUNG wire#w4
   RUNG wire#w4
      Coil( "Safetyinterface".StackDoor7.monitoring.DoorLock )
   END_RUNG
   // the same network as SCL:
   "Safetyinterface".StackDoor7.monitoring.DoorOpen := #TRUE AND ("Safety.DataFromSafety".fDoorCoilStatus.jrWinderDoorOpen OR (NOT "Safety.DataFromSafety".fDoorCoilStatus.jrWinderDoorOpen AND "Safety.DataFromSafety".fDoorDrive.fDoor7.ackReq AND NOT "Global.Data".general.clock.cycle1000Msec AND NOT "Safety.DataFromSafety".fDoorSwitchStatus.jrWinderDoorOpen));
   "Safetyinterface".StackDoor7.monitoring.DoorUnLock := #TRUE AND "Safety.DataFromSafety".fDoorCoilStatus.jrWinderDoorOpen;
   #_w1 := #TRUE AND NOT "Safety.DataFromSafety".fDoorCoilStatus.jrWinderDoorOpen AND (NOT "Safety.DataFromSafety".fDoorDrive.fDoor7.ackReq OR ("Safety.DataFromSafety".fDoorDrive.fDoor7.ackReq AND NOT "Global.Data".general.clock.cycle1000Msec));
   "Safetyinterface".StackDoor7.monitoring.DoorClose := #_w1 AND NOT "Safety.DataFromSafety".fDoorSwitchStatus.jrWinderDoorOpen AND NOT "Safetyinterface".StackDoor7.monitoring.DoorOpen;
   "Safetyinterface".StackDoor7.monitoring.DoorLock := #_w1;
END_REGION

REGION Network 11: At Least One Door Unlock Command
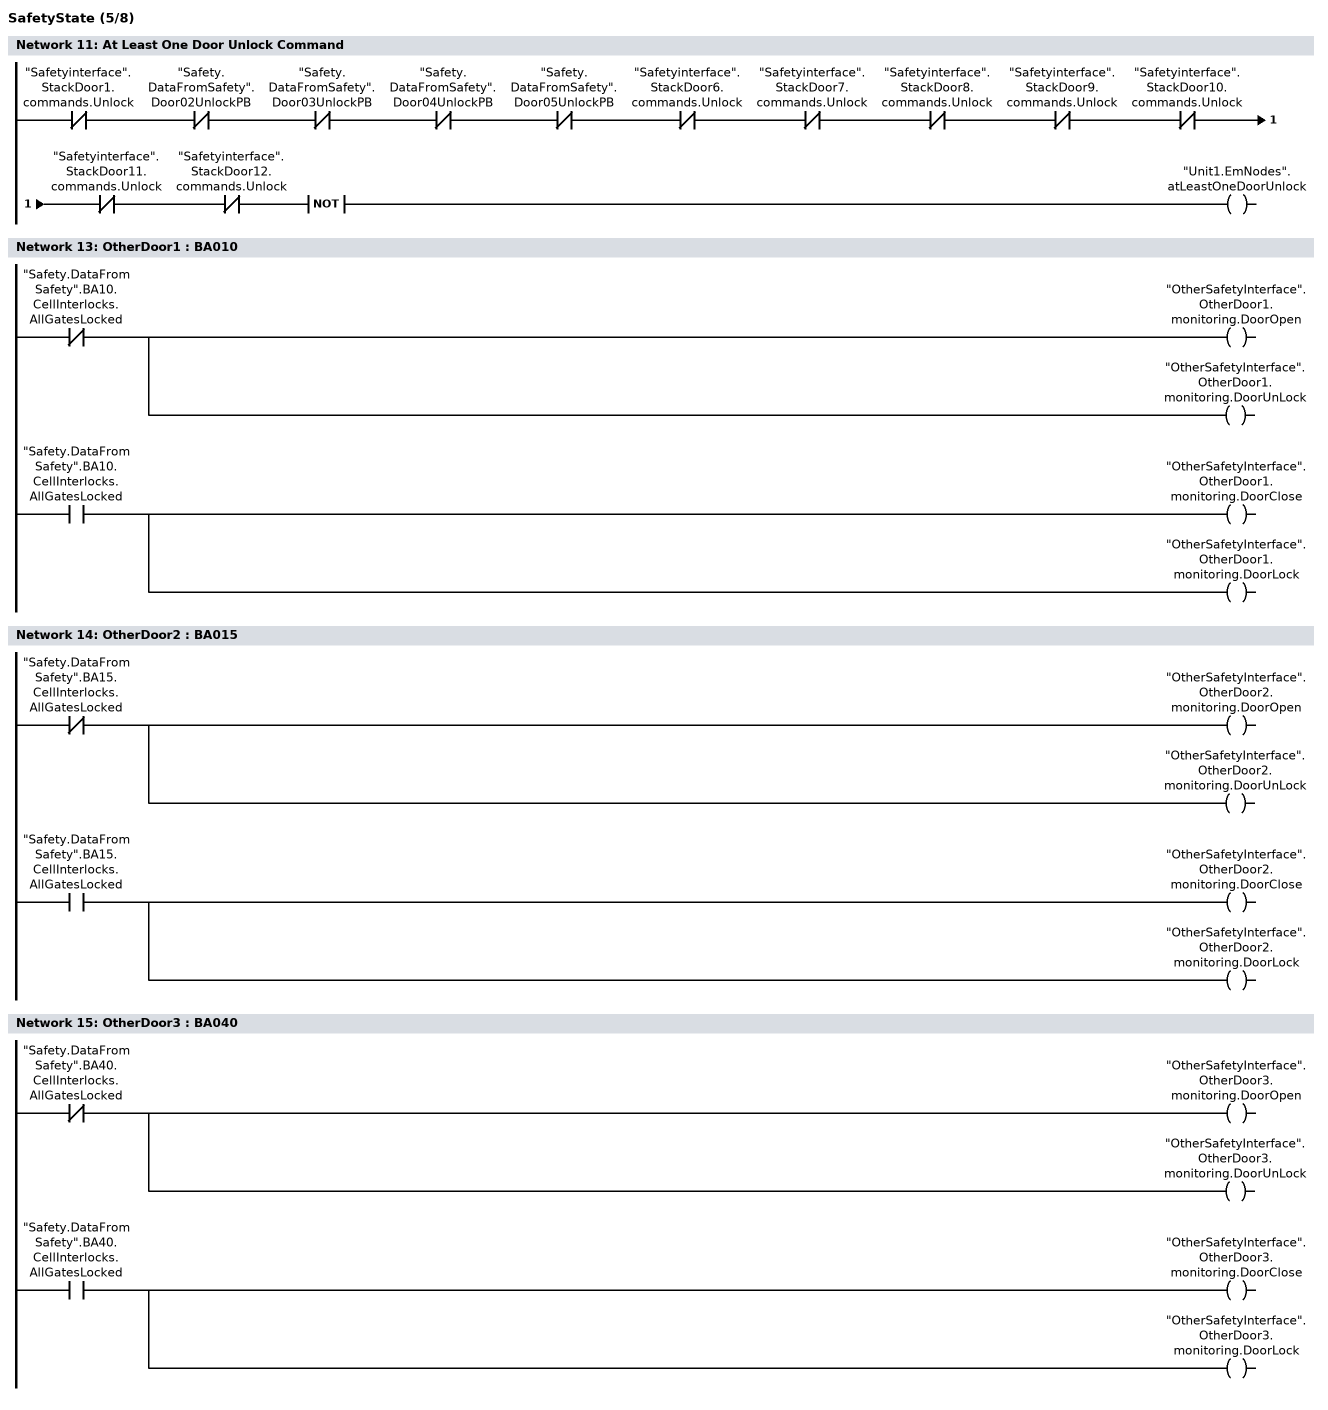
   RUNG wire#powerrail
      I_Contact( "Safetyinterface".StackDoor1.commands.Unlock )
      I_Contact( "Safety.DataFromSafety".Door02UnlockPB )
      I_Contact( "Safety.DataFromSafety".Door03UnlockPB )
      I_Contact( "Safety.DataFromSafety".Door04UnlockPB )
      I_Contact( "Safety.DataFromSafety".Door05UnlockPB )
      I_Contact( "Safetyinterface".StackDoor6.commands.Unlock )
      I_Contact( "Safetyinterface".StackDoor7.commands.Unlock )
      I_Contact( "Safetyinterface".StackDoor8.commands.Unlock )
      I_Contact( "Safetyinterface".StackDoor9.commands.Unlock )
      I_Contact( "Safetyinterface".StackDoor10.commands.Unlock )
      I_Contact( "Safetyinterface".StackDoor11.commands.Unlock )
      I_Contact( "Safetyinterface".StackDoor12.commands.Unlock )
      Not()
      Coil( "Unit1.EmNodes".atLeastOneDoorUnlock )
   END_RUNG
   // the same network as SCL:
   "Unit1.EmNodes".atLeastOneDoorUnlock := NOT (NOT "Safetyinterface".StackDoor1.commands.Unlock AND NOT "Safety.DataFromSafety".Door02UnlockPB AND NOT "Safety.DataFromSafety".Door03UnlockPB AND NOT "Safety.DataFromSafety".Door04UnlockPB AND NOT "Safety.DataFromSafety".Door05UnlockPB AND NOT "Safetyinterface".StackDoor6.commands.Unlock AND NOT "Safetyinterface".StackDoor7.commands.Unlock AND NOT "Safetyinterface".StackDoor8.commands.Unlock AND NOT "Safetyinterface".StackDoor9.commands.Unlock AND NOT "Safetyinterface".StackDoor10.commands.Unlock AND NOT "Safetyinterface".StackDoor11.commands.Unlock AND NOT "Safetyinterface".StackDoor12.commands.Unlock);
END_REGION

REGION Network 12: ***** Other Safety Interface *****
END_REGION

REGION Network 13: OtherDoor1 : BA010
   RUNG wire#powerrail
      I_Contact( "Safety.DataFromSafety".BA10.CellInterlocks.AllGatesLocked )
      wire#w1
      Coil( "OtherSafetyInterface".OtherDoor1.monitoring.DoorOpen )
   END_RUNG
   RUNG wire#w1
      Coil( "OtherSafetyInterface".OtherDoor1.monitoring.DoorUnLock )
   END_RUNG
   RUNG wire#powerrail
      Contact( "Safety.DataFromSafety".BA10.CellInterlocks.AllGatesLocked )
      wire#w2
      Coil( "OtherSafetyInterface".OtherDoor1.monitoring.DoorClose )
   END_RUNG
   RUNG wire#w2
      Coil( "OtherSafetyInterface".OtherDoor1.monitoring.DoorLock )
   END_RUNG
   // the same network as SCL:
   "OtherSafetyInterface".OtherDoor1.monitoring.DoorOpen := NOT "Safety.DataFromSafety".BA10.CellInterlocks.AllGatesLocked;
   "OtherSafetyInterface".OtherDoor1.monitoring.DoorUnLock := NOT "Safety.DataFromSafety".BA10.CellInterlocks.AllGatesLocked;
   "OtherSafetyInterface".OtherDoor1.monitoring.DoorClose := "Safety.DataFromSafety".BA10.CellInterlocks.AllGatesLocked;
   "OtherSafetyInterface".OtherDoor1.monitoring.DoorLock := "Safety.DataFromSafety".BA10.CellInterlocks.AllGatesLocked;
END_REGION

REGION Network 14: OtherDoor2 : BA015
   RUNG wire#powerrail
      I_Contact( "Safety.DataFromSafety".BA15.CellInterlocks.AllGatesLocked )
      wire#w1
      Coil( "OtherSafetyInterface".OtherDoor2.monitoring.DoorOpen )
   END_RUNG
   RUNG wire#w1
      Coil( "OtherSafetyInterface".OtherDoor2.monitoring.DoorUnLock )
   END_RUNG
   RUNG wire#powerrail
      Contact( "Safety.DataFromSafety".BA15.CellInterlocks.AllGatesLocked )
      wire#w2
      Coil( "OtherSafetyInterface".OtherDoor2.monitoring.DoorClose )
   END_RUNG
   RUNG wire#w2
      Coil( "OtherSafetyInterface".OtherDoor2.monitoring.DoorLock )
   END_RUNG
   // the same network as SCL:
   "OtherSafetyInterface".OtherDoor2.monitoring.DoorOpen := NOT "Safety.DataFromSafety".BA15.CellInterlocks.AllGatesLocked;
   "OtherSafetyInterface".OtherDoor2.monitoring.DoorUnLock := NOT "Safety.DataFromSafety".BA15.CellInterlocks.AllGatesLocked;
   "OtherSafetyInterface".OtherDoor2.monitoring.DoorClose := "Safety.DataFromSafety".BA15.CellInterlocks.AllGatesLocked;
   "OtherSafetyInterface".OtherDoor2.monitoring.DoorLock := "Safety.DataFromSafety".BA15.CellInterlocks.AllGatesLocked;
END_REGION

REGION Network 15: OtherDoor3 : BA040
   RUNG wire#powerrail
      I_Contact( "Safety.DataFromSafety".BA40.CellInterlocks.AllGatesLocked )
      wire#w1
      Coil( "OtherSafetyInterface".OtherDoor3.monitoring.DoorOpen )
   END_RUNG
   RUNG wire#w1
      Coil( "OtherSafetyInterface".OtherDoor3.monitoring.DoorUnLock )
   END_RUNG
   RUNG wire#powerrail
      Contact( "Safety.DataFromSafety".BA40.CellInterlocks.AllGatesLocked )
      wire#w2
      Coil( "OtherSafetyInterface".OtherDoor3.monitoring.DoorClose )
   END_RUNG
   RUNG wire#w2
      Coil( "OtherSafetyInterface".OtherDoor3.monitoring.DoorLock )
   END_RUNG
   // the same network as SCL:
   "OtherSafetyInterface".OtherDoor3.monitoring.DoorOpen := NOT "Safety.DataFromSafety".BA40.CellInterlocks.AllGatesLocked;
   "OtherSafetyInterface".OtherDoor3.monitoring.DoorUnLock := NOT "Safety.DataFromSafety".BA40.CellInterlocks.AllGatesLocked;
   "OtherSafetyInterface".OtherDoor3.monitoring.DoorClose := "Safety.DataFromSafety".BA40.CellInterlocks.AllGatesLocked;
   "OtherSafetyInterface".OtherDoor3.monitoring.DoorLock := "Safety.DataFromSafety".BA40.CellInterlocks.AllGatesLocked;
END_REGION

REGION Network 16: OtherDoor4 : BA060
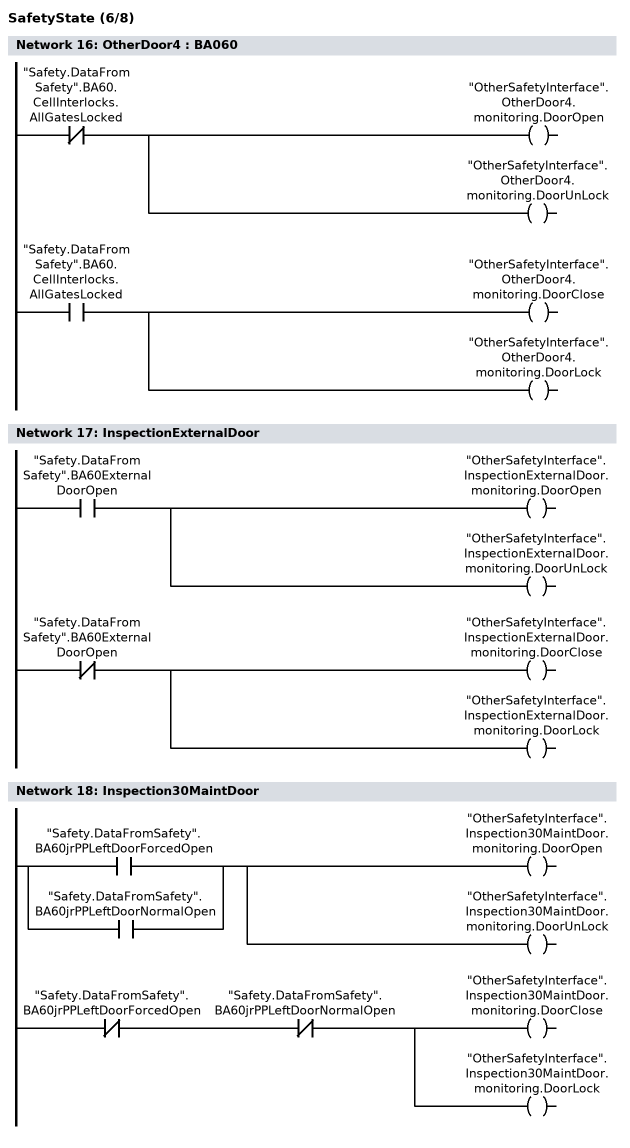
   RUNG wire#powerrail
      I_Contact( "Safety.DataFromSafety".BA60.CellInterlocks.AllGatesLocked )
      wire#w1
      Coil( "OtherSafetyInterface".OtherDoor4.monitoring.DoorOpen )
   END_RUNG
   RUNG wire#w1
      Coil( "OtherSafetyInterface".OtherDoor4.monitoring.DoorUnLock )
   END_RUNG
   RUNG wire#powerrail
      Contact( "Safety.DataFromSafety".BA60.CellInterlocks.AllGatesLocked )
      wire#w2
      Coil( "OtherSafetyInterface".OtherDoor4.monitoring.DoorClose )
   END_RUNG
   RUNG wire#w2
      Coil( "OtherSafetyInterface".OtherDoor4.monitoring.DoorLock )
   END_RUNG
   // the same network as SCL:
   "OtherSafetyInterface".OtherDoor4.monitoring.DoorOpen := NOT "Safety.DataFromSafety".BA60.CellInterlocks.AllGatesLocked;
   "OtherSafetyInterface".OtherDoor4.monitoring.DoorUnLock := NOT "Safety.DataFromSafety".BA60.CellInterlocks.AllGatesLocked;
   "OtherSafetyInterface".OtherDoor4.monitoring.DoorClose := "Safety.DataFromSafety".BA60.CellInterlocks.AllGatesLocked;
   "OtherSafetyInterface".OtherDoor4.monitoring.DoorLock := "Safety.DataFromSafety".BA60.CellInterlocks.AllGatesLocked;
END_REGION

REGION Network 17: InspectionExternalDoor
   RUNG wire#powerrail
      Contact( "Safety.DataFromSafety".BA60ExternalDoorOpen )
      wire#w1
      Coil( "OtherSafetyInterface".InspectionExternalDoor.monitoring.DoorOpen )
   END_RUNG
   RUNG wire#w1
      Coil( "OtherSafetyInterface".InspectionExternalDoor.monitoring.DoorUnLock )
   END_RUNG
   RUNG wire#powerrail
      I_Contact( "Safety.DataFromSafety".BA60ExternalDoorOpen )
      wire#w2
      Coil( "OtherSafetyInterface".InspectionExternalDoor.monitoring.DoorClose )
   END_RUNG
   RUNG wire#w2
      Coil( "OtherSafetyInterface".InspectionExternalDoor.monitoring.DoorLock )
   END_RUNG
   // the same network as SCL:
   "OtherSafetyInterface".InspectionExternalDoor.monitoring.DoorOpen := "Safety.DataFromSafety".BA60ExternalDoorOpen;
   "OtherSafetyInterface".InspectionExternalDoor.monitoring.DoorUnLock := "Safety.DataFromSafety".BA60ExternalDoorOpen;
   "OtherSafetyInterface".InspectionExternalDoor.monitoring.DoorClose := NOT "Safety.DataFromSafety".BA60ExternalDoorOpen;
   "OtherSafetyInterface".InspectionExternalDoor.monitoring.DoorLock := NOT "Safety.DataFromSafety".BA60ExternalDoorOpen;
END_REGION

REGION Network 18: Inspection30MaintDoor
   RUNG wire#powerrail
      Contact( "Safety.DataFromSafety".BA60jrPPLeftDoorForcedOpen )
      wire#w1
      Coil( "OtherSafetyInterface".Inspection30MaintDoor.monitoring.DoorOpen )
   END_RUNG
   RUNG wire#powerrail
      Contact( "Safety.DataFromSafety".BA60jrPPLeftDoorNormalOpen )
   END_RUNG wire#w1
   RUNG wire#w1
      Coil( "OtherSafetyInterface".Inspection30MaintDoor.monitoring.DoorUnLock )
   END_RUNG
   RUNG wire#powerrail
      I_Contact( "Safety.DataFromSafety".BA60jrPPLeftDoorForcedOpen )
      I_Contact( "Safety.DataFromSafety".BA60jrPPLeftDoorNormalOpen )
      wire#w2
      Coil( "OtherSafetyInterface".Inspection30MaintDoor.monitoring.DoorClose )
   END_RUNG
   RUNG wire#w2
      Coil( "OtherSafetyInterface".Inspection30MaintDoor.monitoring.DoorLock )
   END_RUNG
   // the same network as SCL:
   "OtherSafetyInterface".Inspection30MaintDoor.monitoring.DoorOpen := "Safety.DataFromSafety".BA60jrPPLeftDoorForcedOpen OR "Safety.DataFromSafety".BA60jrPPLeftDoorNormalOpen;
   "OtherSafetyInterface".Inspection30MaintDoor.monitoring.DoorUnLock := "OtherSafetyInterface".Inspection30MaintDoor.monitoring.DoorOpen;
   "OtherSafetyInterface".Inspection30MaintDoor.monitoring.DoorClose := NOT "Safety.DataFromSafety".BA60jrPPLeftDoorForcedOpen AND NOT "Safety.DataFromSafety".BA60jrPPLeftDoorNormalOpen;
   "OtherSafetyInterface".Inspection30MaintDoor.monitoring.DoorLock := "OtherSafetyInterface".Inspection30MaintDoor.monitoring.DoorClose;
END_REGION

REGION Network 19: Inspection40MaintDoor
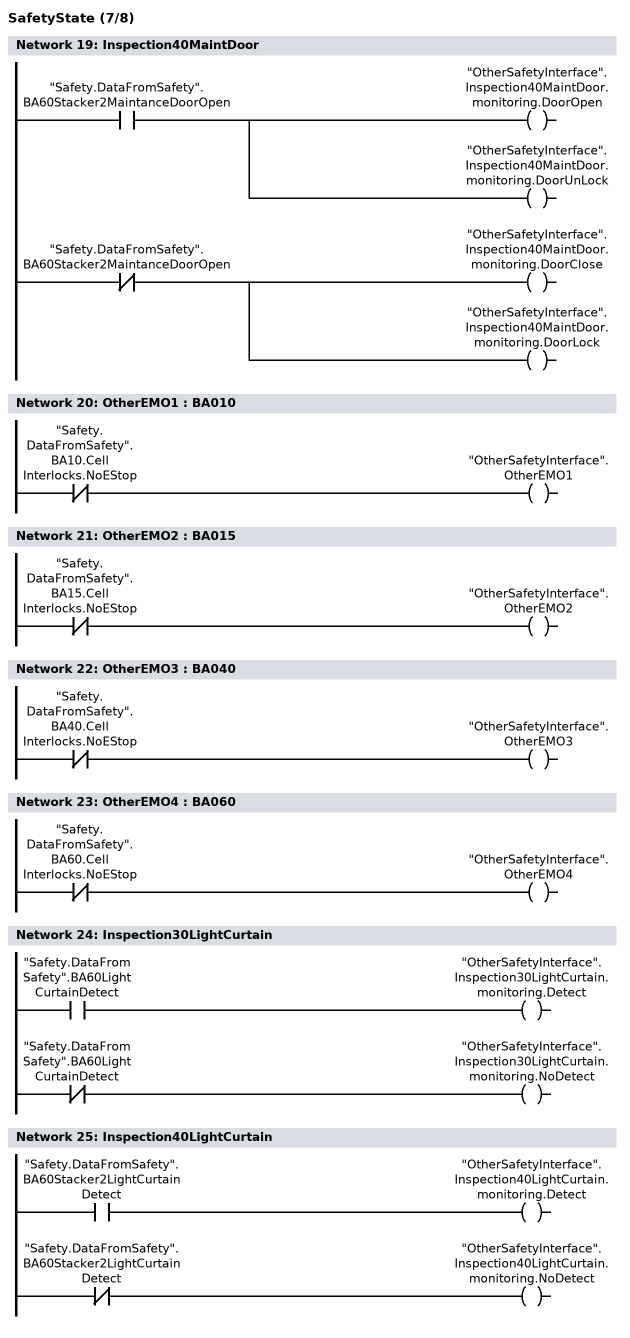
   RUNG wire#powerrail
      Contact( "Safety.DataFromSafety".BA60Stacker2MaintanceDoorOpen )
      wire#w1
      Coil( "OtherSafetyInterface".Inspection40MaintDoor.monitoring.DoorOpen )
   END_RUNG
   RUNG wire#w1
      Coil( "OtherSafetyInterface".Inspection40MaintDoor.monitoring.DoorUnLock )
   END_RUNG
   RUNG wire#powerrail
      I_Contact( "Safety.DataFromSafety".BA60Stacker2MaintanceDoorOpen )
      wire#w2
      Coil( "OtherSafetyInterface".Inspection40MaintDoor.monitoring.DoorClose )
   END_RUNG
   RUNG wire#w2
      Coil( "OtherSafetyInterface".Inspection40MaintDoor.monitoring.DoorLock )
   END_RUNG
   // the same network as SCL:
   "OtherSafetyInterface".Inspection40MaintDoor.monitoring.DoorOpen := "Safety.DataFromSafety".BA60Stacker2MaintanceDoorOpen;
   "OtherSafetyInterface".Inspection40MaintDoor.monitoring.DoorUnLock := "Safety.DataFromSafety".BA60Stacker2MaintanceDoorOpen;
   "OtherSafetyInterface".Inspection40MaintDoor.monitoring.DoorClose := NOT "Safety.DataFromSafety".BA60Stacker2MaintanceDoorOpen;
   "OtherSafetyInterface".Inspection40MaintDoor.monitoring.DoorLock := NOT "Safety.DataFromSafety".BA60Stacker2MaintanceDoorOpen;
END_REGION

REGION Network 20: OtherEMO1 : BA010
   RUNG wire#powerrail
      I_Contact( "Safety.DataFromSafety".BA10.CellInterlocks.NoEStop )
      Coil( "OtherSafetyInterface".OtherEMO1 )
   END_RUNG
   // the same network as SCL:
   "OtherSafetyInterface".OtherEMO1 := NOT "Safety.DataFromSafety".BA10.CellInterlocks.NoEStop;
END_REGION

REGION Network 21: OtherEMO2 : BA015
   RUNG wire#powerrail
      I_Contact( "Safety.DataFromSafety".BA15.CellInterlocks.NoEStop )
      Coil( "OtherSafetyInterface".OtherEMO2 )
   END_RUNG
   // the same network as SCL:
   "OtherSafetyInterface".OtherEMO2 := NOT "Safety.DataFromSafety".BA15.CellInterlocks.NoEStop;
END_REGION

REGION Network 22: OtherEMO3 : BA040
   RUNG wire#powerrail
      I_Contact( "Safety.DataFromSafety".BA40.CellInterlocks.NoEStop )
      Coil( "OtherSafetyInterface".OtherEMO3 )
   END_RUNG
   // the same network as SCL:
   "OtherSafetyInterface".OtherEMO3 := NOT "Safety.DataFromSafety".BA40.CellInterlocks.NoEStop;
END_REGION

REGION Network 23: OtherEMO4 : BA060
   RUNG wire#powerrail
      I_Contact( "Safety.DataFromSafety".BA60.CellInterlocks.NoEStop )
      Coil( "OtherSafetyInterface".OtherEMO4 )
   END_RUNG
   // the same network as SCL:
   "OtherSafetyInterface".OtherEMO4 := NOT "Safety.DataFromSafety".BA60.CellInterlocks.NoEStop;
END_REGION

REGION Network 24: Inspection30LightCurtain
   RUNG wire#powerrail
      Contact( "Safety.DataFromSafety".BA60LightCurtainDetect )
      Coil( "OtherSafetyInterface".Inspection30LightCurtain.monitoring.Detect )
   END_RUNG
   RUNG wire#powerrail
      I_Contact( "Safety.DataFromSafety".BA60LightCurtainDetect )
      Coil( "OtherSafetyInterface".Inspection30LightCurtain.monitoring.NoDetect )
   END_RUNG
   // the same network as SCL:
   "OtherSafetyInterface".Inspection30LightCurtain.monitoring.Detect := "Safety.DataFromSafety".BA60LightCurtainDetect;
   "OtherSafetyInterface".Inspection30LightCurtain.monitoring.NoDetect := NOT "Safety.DataFromSafety".BA60LightCurtainDetect;
END_REGION

REGION Network 25: Inspection40LightCurtain
   RUNG wire#powerrail
      Contact( "Safety.DataFromSafety".BA60Stacker2LightCurtainDetect )
      Coil( "OtherSafetyInterface".Inspection40LightCurtain.monitoring.Detect )
   END_RUNG
   RUNG wire#powerrail
      I_Contact( "Safety.DataFromSafety".BA60Stacker2LightCurtainDetect )
      Coil( "OtherSafetyInterface".Inspection40LightCurtain.monitoring.NoDetect )
   END_RUNG
   // the same network as SCL:
   "OtherSafetyInterface".Inspection40LightCurtain.monitoring.Detect := "Safety.DataFromSafety".BA60Stacker2LightCurtainDetect;
   "OtherSafetyInterface".Inspection40LightCurtain.monitoring.NoDetect := NOT "Safety.DataFromSafety".BA60Stacker2LightCurtainDetect;
END_REGION

REGION Network 26: 30CathodeConveyorCover
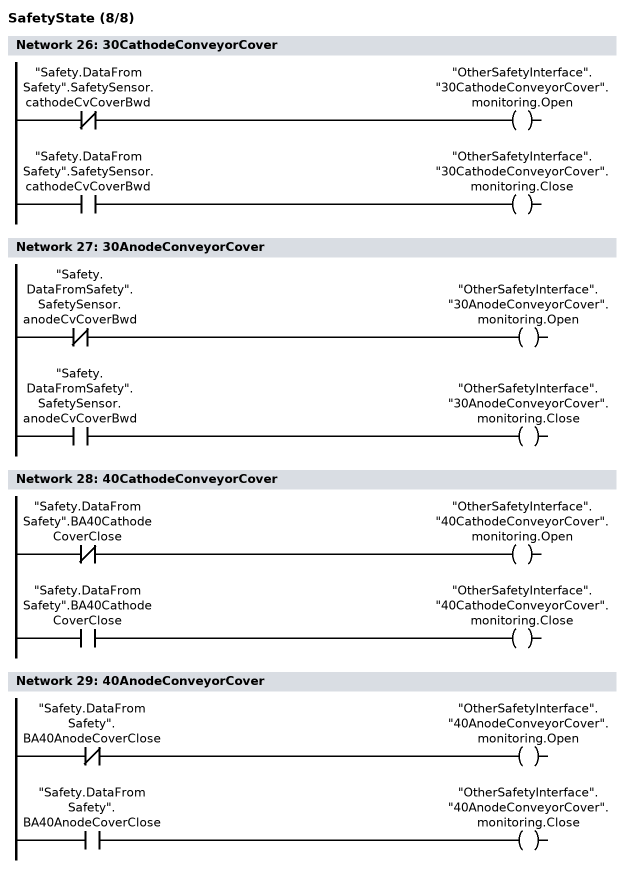
   RUNG wire#powerrail
      I_Contact( "Safety.DataFromSafety".SafetySensor.cathodeCvCoverBwd )
      Coil( "OtherSafetyInterface"."30CathodeConveyorCover".monitoring.Open )
   END_RUNG
   RUNG wire#powerrail
      Contact( "Safety.DataFromSafety".SafetySensor.cathodeCvCoverBwd )
      Coil( "OtherSafetyInterface"."30CathodeConveyorCover".monitoring.Close )
   END_RUNG
   // the same network as SCL:
   "OtherSafetyInterface"."30CathodeConveyorCover".monitoring.Open := NOT "Safety.DataFromSafety".SafetySensor.cathodeCvCoverBwd;
   "OtherSafetyInterface"."30CathodeConveyorCover".monitoring.Close := "Safety.DataFromSafety".SafetySensor.cathodeCvCoverBwd;
END_REGION

REGION Network 27: 30AnodeConveyorCover
   RUNG wire#powerrail
      I_Contact( "Safety.DataFromSafety".SafetySensor.anodeCvCoverBwd )
      Coil( "OtherSafetyInterface"."30AnodeConveyorCover".monitoring.Open )
   END_RUNG
   RUNG wire#powerrail
      Contact( "Safety.DataFromSafety".SafetySensor.anodeCvCoverBwd )
      Coil( "OtherSafetyInterface"."30AnodeConveyorCover".monitoring.Close )
   END_RUNG
   // the same network as SCL:
   "OtherSafetyInterface"."30AnodeConveyorCover".monitoring.Open := NOT "Safety.DataFromSafety".SafetySensor.anodeCvCoverBwd;
   "OtherSafetyInterface"."30AnodeConveyorCover".monitoring.Close := "Safety.DataFromSafety".SafetySensor.anodeCvCoverBwd;
END_REGION

REGION Network 28: 40CathodeConveyorCover
   RUNG wire#powerrail
      I_Contact( "Safety.DataFromSafety".BA40CathodeCoverClose )
      Coil( "OtherSafetyInterface"."40CathodeConveyorCover".monitoring.Open )
   END_RUNG
   RUNG wire#powerrail
      Contact( "Safety.DataFromSafety".BA40CathodeCoverClose )
      Coil( "OtherSafetyInterface"."40CathodeConveyorCover".monitoring.Close )
   END_RUNG
   // the same network as SCL:
   "OtherSafetyInterface"."40CathodeConveyorCover".monitoring.Open := NOT "Safety.DataFromSafety".BA40CathodeCoverClose;
   "OtherSafetyInterface"."40CathodeConveyorCover".monitoring.Close := "Safety.DataFromSafety".BA40CathodeCoverClose;
END_REGION

REGION Network 29: 40AnodeConveyorCover
   RUNG wire#powerrail
      I_Contact( "Safety.DataFromSafety".BA40AnodeCoverClose )
      Coil( "OtherSafetyInterface"."40AnodeConveyorCover".monitoring.Open )
   END_RUNG
   RUNG wire#powerrail
      Contact( "Safety.DataFromSafety".BA40AnodeCoverClose )
      Coil( "OtherSafetyInterface"."40AnodeConveyorCover".monitoring.Close )
   END_RUNG
   // the same network as SCL:
   "OtherSafetyInterface"."40AnodeConveyorCover".monitoring.Open := NOT "Safety.DataFromSafety".BA40AnodeCoverClose;
   "OtherSafetyInterface"."40AnodeConveyorCover".monitoring.Close := "Safety.DataFromSafety".BA40AnodeCoverClose;
END_REGION
END_FUNCTION

FUNCTION "ReadMe02" : Void
{ S7_Optimized_Access := 'TRUE' ; Published := 'FALSE' }
VERSION : 0.1

BEGIN
	// The folder structure of the software unit CentralFunctions correlates with the main navigation in the HMI.
	// For easier orientation, all folders are listed, but some are empty because there is no PLC logic needed, there is only content on the HMI side.
	// Any PLC logic that should relate to the screens on the HMI for that chapter can be added in this folder.
END_FUNCTION

FUNCTION "CallManualOperationLineStartup" : Void
{ S7_Optimized_Access := 'TRUE' ; Published := 'FALSE' }
VERSION : 0.1

BEGIN
	REGION Description
	(*
	    Startup call to set the configuration of the Manual Operation Line for the Equipment modules
	*)
	    
	END_REGION
	
	"LAF_InternalManual".emsWithManualOpConfigured.maxNoOfEms := "NO_OF_EM";
	
	REGION Unit 1 Equipment Module 0 configuration
	    "ManualOperationControl_U1Em0".manualOperationEm.equipmentModuleNum := 1010;
	    "ManualOperationControl_U1Em0".manualOperationEmArea[2].displayedLines := '6;';
	    "ManualOperationControl_U1Em0".manualOperationEmArea[1].displayedLines := '21;';
	END_REGION
	
	REGION Unit 1 Equipment Module 1 configuration
	    "ManualOperationControl_U1Em1".manualOperationEm.equipmentModuleNum := 1020;
	    "ManualOperationControl_U1Em1".manualOperationEmArea[2].displayedLines := '6;';
	    "ManualOperationControl_U1Em1".manualOperationEmArea[1].displayedLines := '21;';
	END_REGION
	
	REGION Unit 1 Equipment Module 2 configuration
	    "ManualOperationControl_U1Em2".manualOperationEm.equipmentModuleNum := 1030;
	    "ManualOperationControl_U1Em2".manualOperationEmArea[2].displayedLines := '1;';
	    "ManualOperationControl_U1Em2".manualOperationEmArea[1].displayedLines := '21-33;';
	END_REGION
	
	REGION Unit 1 Equipment Module 3 configuration
	    "ManualOperationControl_U1Em3".manualOperationEm.equipmentModuleNum := 1040;
	    "ManualOperationControl_U1Em3".manualOperationEmArea[2].displayedLines := '6-7;';
	    "ManualOperationControl_U1Em3".manualOperationEmArea[1].displayedLines := '21-24;';
	END_REGION
	
	REGION Unit 1 Equipment Module 4 configuration
	    "ManualOperationControl_U1Em4".manualOperationEm.equipmentModuleNum := 1050;
	    "ManualOperationControl_U1Em4".manualOperationEmArea[2].displayedLines := '6-13;';
	    "ManualOperationControl_U1Em4".manualOperationEmArea[1].displayedLines := '21-33;';
	END_REGION
	
	REGION Unit 1 Equipment Module 5 configuration
	    "ManualOperationControl_U1Em5".manualOperationEm.equipmentModuleNum := 1060;
	    "ManualOperationControl_U1Em5".manualOperationEmArea[2].displayedLines := '6-13;';
	    "ManualOperationControl_U1Em5".manualOperationEmArea[1].displayedLines := '21-33;';
	END_REGION
	
	REGION Unit 1 Equipment Module 6 configuration
	    "ManualOperationControl_U1Em6".manualOperationEm.equipmentModuleNum := 1070;
	    "ManualOperationControl_U1Em6".manualOperationEmArea[2].displayedLines := '6-18;';
	    "ManualOperationControl_U1Em6".manualOperationEmArea[1].displayedLines := '21-26;';
	END_REGION
	
	REGION Unit 1 Equipment Module 7 configuration
	    "ManualOperationControl_U1Em7".manualOperationEm.equipmentModuleNum := 1080;
	    "ManualOperationControl_U1Em7".manualOperationEmArea[2].displayedLines := '6-14;';
	    "ManualOperationControl_U1Em7".manualOperationEmArea[1].displayedLines := '21-30;';
	END_REGION
	
	REGION CITI EM1 configuration
	    // Statement section REGION
	    "ManualOperationControl_CITIEm1".manualOperationEm.equipmentModuleNum := 5010;
	    "ManualOperationControl_CITIEm1".manualOperationEmArea[2].displayedLines := '1-5;';
	END_REGION
	
END_FUNCTION

FUNCTION_BLOCK "GetIdentMv"
{ S7_Optimized_Access := 'TRUE' ; Published := 'TRUE' }
VERSION : 0.1
   VAR_INPUT 
      identMvAllUnits { ExternalAccessible := 'False'; ExternalVisible := 'False'; ExternalWritable := 'False'} : Array[0.."NO_OF_UNITS"] of "typeEMIdentMv";   // HMI: motorstarter values
      numberOfMvReaders : USInt;
   END_VAR

   VAR_OUTPUT 
      selectedUnit : USInt;
      selectedEM : USInt;
      error : Word;
   END_VAR

   VAR_IN_OUT 
      IdentMvInterfaceHmi : "typeIdentMvHmi";
   END_VAR

   VAR 
      statSelectedEMIdentMv : USInt := 1;
      statSelectedUnitIdentRMv : USInt := 1;   // HMI: Selected unit
   END_VAR

   VAR_TEMP 
      tempEnable : Bool;   // Temporary value for input 'enable'
      tempMvReader : Array[0.."NO_OF_MV_IDENT_DEVICES"] of "LSicar_typeIdentInterfaceHmi";
      tempIndexIdentMv : USInt;
      tempNoOfidertMv : USInt;
   END_VAR

   VAR CONSTANT 
      "INVALID UNIT" : Word := 16#7001;   // non existant unit
      "INVALID EM" : Word := 16#7002;   // non existant em
      OK : Word := 16#7000;
   END_VAR


BEGIN
	REGION BLOCK INFO HEADER
	    //===============================================================================
	    // Siemens AG / (c)Copyright 2024
	    //-------------------------------------------------------------------------------
	    // Title:            LAF_GetMotorstarterSignals
	    // Comment/Function: This block reads diagnostic information of a Motorstarter depending
	    //                   on the unit and Control Module selected in the HMI by the user.
	    // Library/Family:   Automation Framework / Motorstarter Diagnostic
	    // Author:           Siemens Digital Industries
	    // Tested with:      S7-1517TF V3.1
	    // Engineering:      TIA Portal V19
	    // Restrictions:     
	    //                   Required UDTs: LAF_typeDriveDiagConfig, LAF_typeDriveDiagInterfaceHmi
	    // Requirements:     S7-1500(T), MC_Version V8.0
	    //-------------------------------------------------------------------------------
	    // Change log table:
	    // Version  | Date       | Expert in charge        | Changes applied
	    //----------|------------|-------------------------|-----------------------------
	    // 01.00.00 | 05.06.2024 | SIMATIC Systems Support | First released version
	    //===============================================================================
	END_REGION BLOCK INFO HEADER
	
	REGION DESCRIPTION
	(/*
	This block reads diagnostic information (control inputs and outputs) of a Motorstarter. 
	At runtime, this block is enabled when the ET200SP Motorstarter screen is shown in the HMI. 
	Based on the selected motorstarter object in the HMI by the user. The shown information in the HMI depends on the
	Unit and Cotrol Module selected. 
	*/)
	END_REGION DESCRIPTION
	
	REGION INPUTS
	    //working with static values to keep the last selected value when opening for the first time the screen  
	  
	    #statSelectedUnitIdentRMv := #IdentMvInterfaceHmi.selectedUnit;
	    #statSelectedEMIdentMv := #IdentMvInterfaceHmi.selectedEM;
	
	END_REGION INPUTS
	
	REGION ASSIGNING TEMPORARY VALUES
	    // Statement section REGION
	    IF #statSelectedUnitIdentRMv <= "NO_OF_UNITS" THEN
	        IF #statSelectedEMIdentMv < "NO_OF_EM" THEN
	            #tempMvReader := #identMvAllUnits[#statSelectedUnitIdentRMv].identMvEM[#statSelectedEMIdentMv].mvReader;
	            #tempNoOfidertMv := #numberOfMvReaders;
	            #error := #OK;
	        ELSE
	            #error := #"INVALID EM";
	        END_IF;
	
	    ELSE
	        #error := #"INVALID UNIT";
	    END_IF;
	
	
	END_REGION
	
	
	REGION OUTPUTS
	    // Statement section REGION
	    #IdentMvInterfaceHmi.mvReader := #tempMvReader;
	    #selectedEM := #statSelectedEMIdentMv;
	    #selectedUnit := #statSelectedUnitIdentRMv;
	END_REGION
	
	
END_FUNCTION_BLOCK

DATA_BLOCK "instTeachingPosCathodeAlignTableAxisY1"   // DB463
// stored: InstanceOfName LER_TeachingPos_Interface, InstanceOfType FB
"LER_TeachingPos_Interface"
   // VAR_INPUT
   //    enable : Bool;
   //    selectTeachingPos : SInt;
   //    indexTeachingPos : SInt;
   // END_VAR
   // VAR_IN_OUT
   //    configurationSetPositions : Array[0..15] of "LBC_typeAxis64PosSetPosition";
   //    moduleInterface : "LBC_typeAxis64PosInterface";
   //    hmiInterface : Array[0..48] of "LER_TypeTeachingPosInterface";
   // END_VAR
   // VAR
   //    statPulse : Array[0..9] of Bool;
   //    statTonTimer : Array[0..15] of TON_TIME;
   //    statLastTeachingPosIndex : SInt;
   // END_VAR
BEGIN
END_DATA_BLOCK

DATA_BLOCK "instTeachingPosCathodeMainPnP1AxisY"   // DB353
// stored: InstanceOfName LER_TeachingPos_Interface, InstanceOfType FB
"LER_TeachingPos_Interface"
   // VAR_INPUT
   //    enable : Bool;
   //    selectTeachingPos : SInt;
   //    indexTeachingPos : SInt;
   // END_VAR
   // VAR_IN_OUT
   //    configurationSetPositions : Array[0..15] of "LBC_typeAxis64PosSetPosition";
   //    moduleInterface : "LBC_typeAxis64PosInterface";
   //    hmiInterface : Array[0..48] of "LER_TypeTeachingPosInterface";
   // END_VAR
   // VAR
   //    statPulse : Array[0..9] of Bool;
   //    statTonTimer : Array[0..15] of TON_TIME;
   //    statLastTeachingPosIndex : SInt;
   // END_VAR
BEGIN
END_DATA_BLOCK

DATA_BLOCK "instTeachingPosCathodeMainPnP2AxisX"   // DB352
// stored: InstanceOfName LER_TeachingPos_Interface, InstanceOfType FB
"LER_TeachingPos_Interface"
   // VAR_INPUT
   //    enable : Bool;
   //    selectTeachingPos : SInt;
   //    indexTeachingPos : SInt;
   // END_VAR
   // VAR_IN_OUT
   //    configurationSetPositions : Array[0..15] of "LBC_typeAxis64PosSetPosition";
   //    moduleInterface : "LBC_typeAxis64PosInterface";
   //    hmiInterface : Array[0..48] of "LER_TypeTeachingPosInterface";
   // END_VAR
   // VAR
   //    statPulse : Array[0..9] of Bool;
   //    statTonTimer : Array[0..15] of TON_TIME;
   //    statLastTeachingPosIndex : SInt;
   // END_VAR
BEGIN
END_DATA_BLOCK

DATA_BLOCK "instTeachingPosFinalRollerFrontAxisX"   // DB465
// stored: InstanceOfName LER_TeachingPos_Interface, InstanceOfType FB
"LER_TeachingPos_Interface"
   // VAR_INPUT
   //    enable : Bool;
   //    selectTeachingPos : SInt;
   //    indexTeachingPos : SInt;
   // END_VAR
   // VAR_IN_OUT
   //    configurationSetPositions : Array[0..15] of "LBC_typeAxis64PosSetPosition";
   //    moduleInterface : "LBC_typeAxis64PosInterface";
   //    hmiInterface : Array[0..48] of "LER_TypeTeachingPosInterface";
   // END_VAR
   // VAR
   //    statPulse : Array[0..9] of Bool;
   //    statTonTimer : Array[0..15] of TON_TIME;
   //    statLastTeachingPosIndex : SInt;
   // END_VAR
BEGIN
END_DATA_BLOCK

DATA_BLOCK "instTeachingPosJRPusherAxisZ"   // DB498
// stored: InstanceOfName LER_TeachingPos_Interface, InstanceOfType FB
"LER_TeachingPos_Interface"
   // VAR_INPUT
   //    enable : Bool;
   //    selectTeachingPos : SInt;
   //    indexTeachingPos : SInt;
   // END_VAR
   // VAR_IN_OUT
   //    configurationSetPositions : Array[0..15] of "LBC_typeAxis64PosSetPosition";
   //    moduleInterface : "LBC_typeAxis64PosInterface";
   //    hmiInterface : Array[0..48] of "LER_TypeTeachingPosInterface";
   // END_VAR
   // VAR
   //    statPulse : Array[0..9] of Bool;
   //    statTonTimer : Array[0..15] of TON_TIME;
   //    statLastTeachingPosIndex : SInt;
   // END_VAR
BEGIN
END_DATA_BLOCK

DATA_BLOCK "instTeachingPosJRWinderFrontAxisY"   // DB484
// stored: InstanceOfName LER_TeachingPos_Interface, InstanceOfType FB
"LER_TeachingPos_Interface"
   // VAR_INPUT
   //    enable : Bool;
   //    selectTeachingPos : SInt;
   //    indexTeachingPos : SInt;
   // END_VAR
   // VAR_IN_OUT
   //    configurationSetPositions : Array[0..15] of "LBC_typeAxis64PosSetPosition";
   //    moduleInterface : "LBC_typeAxis64PosInterface";
   //    hmiInterface : Array[0..48] of "LER_TypeTeachingPosInterface";
   // END_VAR
   // VAR
   //    statPulse : Array[0..9] of Bool;
   //    statTonTimer : Array[0..15] of TON_TIME;
   //    statLastTeachingPosIndex : SInt;
   // END_VAR
BEGIN
END_DATA_BLOCK

DATA_BLOCK "instTeachingPosMendrelAnodeRearAxisZ"   // DB470
// stored: InstanceOfName LER_TeachingPos_Interface, InstanceOfType FB
"LER_TeachingPos_Interface"
   // VAR_INPUT
   //    enable : Bool;
   //    selectTeachingPos : SInt;
   //    indexTeachingPos : SInt;
   // END_VAR
   // VAR_IN_OUT
   //    configurationSetPositions : Array[0..15] of "LBC_typeAxis64PosSetPosition";
   //    moduleInterface : "LBC_typeAxis64PosInterface";
   //    hmiInterface : Array[0..48] of "LER_TypeTeachingPosInterface";
   // END_VAR
   // VAR
   //    statPulse : Array[0..9] of Bool;
   //    statTonTimer : Array[0..15] of TON_TIME;
   //    statLastTeachingPosIndex : SInt;
   // END_VAR
BEGIN
END_DATA_BLOCK

DATA_BLOCK "instTeachingPosSepaGripperAxisZ"   // DB481
// stored: InstanceOfName LER_TeachingPos_Interface, InstanceOfType FB
"LER_TeachingPos_Interface"
   // VAR_INPUT
   //    enable : Bool;
   //    selectTeachingPos : SInt;
   //    indexTeachingPos : SInt;
   // END_VAR
   // VAR_IN_OUT
   //    configurationSetPositions : Array[0..15] of "LBC_typeAxis64PosSetPosition";
   //    moduleInterface : "LBC_typeAxis64PosInterface";
   //    hmiInterface : Array[0..48] of "LER_TypeTeachingPosInterface";
   // END_VAR
   // VAR
   //    statPulse : Array[0..9] of Bool;
   //    statTonTimer : Array[0..15] of TON_TIME;
   //    statLastTeachingPosIndex : SInt;
   // END_VAR
BEGIN
END_DATA_BLOCK

DATA_BLOCK "instTeachingPosStackTableOutFrontAxisZ"   // DB476
// stored: InstanceOfName LER_TeachingPos_Interface, InstanceOfType FB
"LER_TeachingPos_Interface"
   // VAR_INPUT
   //    enable : Bool;
   //    selectTeachingPos : SInt;
   //    indexTeachingPos : SInt;
   // END_VAR
   // VAR_IN_OUT
   //    configurationSetPositions : Array[0..15] of "LBC_typeAxis64PosSetPosition";
   //    moduleInterface : "LBC_typeAxis64PosInterface";
   //    hmiInterface : Array[0..48] of "LER_TypeTeachingPosInterface";
   // END_VAR
   // VAR
   //    statPulse : Array[0..9] of Bool;
   //    statTonTimer : Array[0..15] of TON_TIME;
   //    statLastTeachingPosIndex : SInt;
   // END_VAR
BEGIN
END_DATA_BLOCK

DATA_BLOCK "instTeachingPosStackTableZ"   // DB475
// stored: InstanceOfName LER_TeachingPos_Interface, InstanceOfType FB
"LER_TeachingPos_Interface"
   // VAR_INPUT
   //    enable : Bool;
   //    selectTeachingPos : SInt;
   //    indexTeachingPos : SInt;
   // END_VAR
   // VAR_IN_OUT
   //    configurationSetPositions : Array[0..15] of "LBC_typeAxis64PosSetPosition";
   //    moduleInterface : "LBC_typeAxis64PosInterface";
   //    hmiInterface : Array[0..48] of "LER_TypeTeachingPosInterface";
   // END_VAR
   // VAR
   //    statPulse : Array[0..9] of Bool;
   //    statTonTimer : Array[0..15] of TON_TIME;
   //    statLastTeachingPosIndex : SInt;
   // END_VAR
BEGIN
END_DATA_BLOCK

DATA_BLOCK "instTeachingPosUnwinderBottomAxisB"   // DB269
// stored: InstanceOfName LER_TeachingPos_Interface, InstanceOfType FB
"LER_TeachingPos_Interface"
   // VAR_INPUT
   //    enable : Bool;
   //    selectTeachingPos : SInt;
   //    indexTeachingPos : SInt;
   // END_VAR
   // VAR_IN_OUT
   //    configurationSetPositions : Array[0..15] of "LBC_typeAxis64PosSetPosition";
   //    moduleInterface : "LBC_typeAxis64PosInterface";
   //    hmiInterface : Array[0..48] of "LER_TypeTeachingPosInterface";
   // END_VAR
   // VAR
   //    statPulse : Array[0..9] of Bool;
   //    statTonTimer : Array[0..15] of TON_TIME;
   //    statLastTeachingPosIndex : SInt;
   // END_VAR
BEGIN
END_DATA_BLOCK

DATA_BLOCK "instTeachingPosUnwinderTopAxisB"   // DB268
// stored: InstanceOfName LER_TeachingPos_Interface, InstanceOfType FB
"LER_TeachingPos_Interface"
   // VAR_INPUT
   //    enable : Bool;
   //    selectTeachingPos : SInt;
   //    indexTeachingPos : SInt;
   // END_VAR
   // VAR_IN_OUT
   //    configurationSetPositions : Array[0..15] of "LBC_typeAxis64PosSetPosition";
   //    moduleInterface : "LBC_typeAxis64PosInterface";
   //    hmiInterface : Array[0..48] of "LER_TypeTeachingPosInterface";
   // END_VAR
   // VAR
   //    statPulse : Array[0..9] of Bool;
   //    statTonTimer : Array[0..15] of TON_TIME;
   //    statLastTeachingPosIndex : SInt;
   // END_VAR
BEGIN
END_DATA_BLOCK

DATA_BLOCK "InstGetSinaEpos"   // DB86
AUTHOR : Siemens Digital Industries
FAMILY : LAF
NAME : LAF_GetSinaEpos
VERSION : 1.1
// stored: InstanceOfName LAF_GetSinaEpos, InstanceOfType FB
"LAF_GetSinaEpos"
   // VAR_INPUT
   //    enable : Bool := TRUE;
   // END_VAR
   // VAR_OUTPUT
   //    valid { ExternalWritable := 'False'} : Bool := FALSE;
   //    busy { ExternalWritable := 'False'} : Bool := FALSE;
   //    error { ExternalWritable := 'False'} : Bool := FALSE;
   //    status { ExternalWritable := 'False'} : Word := 16#7000;
   //    diagnostics { ExternalWritable := 'False'} : "LAF_typeDiagnostics";
   //    statusWriteRecord { ExternalAccessible := 'False'; ExternalVisible := 'False'; ExternalWritable := 'False'} : DWord := 16#0000_0000;
   //    statusReadRecord { ExternalAccessible := 'False'; ExternalVisible := 'False'; ExternalWritable := 'False'} : DWord := 16#0000_0000;
   // END_VAR
   // VAR_IN_OUT
   //    configuration : Array[*] of "LAF_typeDriveDiagConfig";
   //    moduleInterface : "LAF_typeDriveDiagInterfaceHmi";
   // END_VAR
   // VAR
   //    statInternal { ExternalAccessible := 'False'; ExternalVisible := 'False'; ExternalWritable := 'False'} : Struct
   //       enablePrevious : Bool := FALSE;
   //       valid : Bool := FALSE;
   //       busy : Bool := FALSE;
   //       error : Bool := FALSE;
   //       errorUserCleared : Bool := FALSE;
   //       errorAutoCleared : Bool := FALSE;
   //       disablingCompleted : Bool := FALSE;
   //       diagnostics : "LAF_typeDiagnostics";
   //       emptyDiagnostics : "LAF_typeDiagnostics";
   //    END_STRUCT;
   //    statMainState { ExternalAccessible := 'False'; ExternalVisible := 'False'; ExternalWritable := 'False'} : DInt := 0;
   //    statArrayMin { ExternalAccessible := 'False'; ExternalVisible := 'False'; ExternalWritable := 'False'} : DInt := 0;
   //    statArrayMax { ExternalAccessible := 'False'; ExternalVisible := 'False'; ExternalWritable := 'False'} : DInt := 0;
   //    instWriteRecord { ExternalAccessible := 'False'; ExternalVisible := 'False'; ExternalWritable := 'False'} : WRREC;
   //    instReadRecord { ExternalAccessible := 'False'; ExternalVisible := 'False'; ExternalWritable := 'False'} : RDREC;
   //    statWriteReq { ExternalAccessible := 'False'; ExternalVisible := 'False'; ExternalWritable := 'False'} : Struct
   //       header : Struct
   //          reqRef : Byte := 16#00;
   //          reqID : Byte := 16#00;
   //          axis : Byte := 16#01;
   //          noPara : Byte := 16#01;
   //       END_STRUCT;
   //       data : Array[0..235] of Byte;
   //    END_STRUCT;
   //    statReadReq { ExternalAccessible := 'False'; ExternalVisible := 'False'; ExternalWritable := 'False'} : Struct
   //       header : Struct
   //          reqRef : Byte := 16#00;
   //          reqID : Byte := 16#00;
   //          axis : Byte := 16#01;
   //          noPara : Byte := 16#01;
   //       END_STRUCT;
   //       data : Array[0..235] of Byte;
   //    END_STRUCT;
   //    instActTimer { ExternalAccessible := 'False'; ExternalVisible := 'False'; ExternalWritable := 'False'} : IEC_TIMER;
   //    instReqTimer { ExternalAccessible := 'False'; ExternalVisible := 'False'; ExternalWritable := 'False'} : IEC_TIMER;
   //    statDataTransRun { ExternalAccessible := 'False'; ExternalVisible := 'False'; ExternalWritable := 'False'} : Bool := FALSE;
   //    statWriteReqSet { ExternalAccessible := 'False'; ExternalVisible := 'False'; ExternalWritable := 'False'} : Bool := FALSE;
   //    statActTimerIn { ExternalAccessible := 'False'; ExternalVisible := 'False'; ExternalWritable := 'False'} : Bool := FALSE;
   //    statPrevTimeValue { ExternalAccessible := 'False'; ExternalVisible := 'False'; ExternalWritable := 'False'} : Time := T#0MS;
   //    statActTimerValueAct { ExternalAccessible := 'False'; ExternalVisible := 'False'; ExternalWritable := 'False'} : Time := T#0MS;
   //    statActTimerValueReq { ExternalAccessible := 'False'; ExternalVisible := 'False'; ExternalWritable := 'False'} : Time := T#0MS;
   //    statPrevDriveIndex { ExternalAccessible := 'False'; ExternalVisible := 'False'; ExternalWritable := 'False'} : DInt := 0;
   // END_VAR
BEGIN
   diagnostics.status := 16#0000;
   diagnostics.subfunctionStatus := 16#0000;
   diagnostics.stateNumber := 0;
   statInternal.diagnostics.status := 16#7000;
   statInternal.diagnostics.subfunctionStatus := 16#0000;
   statInternal.diagnostics.stateNumber := 0;
   statInternal.emptyDiagnostics.status := 16#7000;
   statInternal.emptyDiagnostics.subfunctionStatus := 16#0000;
   statInternal.emptyDiagnostics.stateNumber := 0;
   instWriteRecord.REQ := FALSE;
   instWriteRecord.ID := 0;
   instWriteRecord.INDEX := 0;
   instWriteRecord.LEN := 0;
   instWriteRecord.DONE := FALSE;
   instWriteRecord.BUSY := FALSE;
   instWriteRecord.ERROR := FALSE;
   instWriteRecord.STATUS := 16#0000_0000;
   instReadRecord.REQ := FALSE;
   instReadRecord.ID := 0;
   instReadRecord.INDEX := 0;
   instReadRecord.MLEN := 0;
   instReadRecord.VALID := FALSE;
   instReadRecord.BUSY := FALSE;
   instReadRecord.ERROR := FALSE;
   instReadRecord.STATUS := 16#0000_0000;
   instReadRecord.LEN := 0;
   statWriteReq.data[0..235] := 16#00;
   statReadReq.data[0..235] := 16#00;
   instActTimer.PT := T#0MS;
   instActTimer.IN := FALSE;
   instReqTimer.PT := T#0MS;
   instReqTimer.IN := FALSE;
END_DATA_BLOCK

